// State machine for decision point
CASE eDecisionPointState OF
	E_DecisionPointState.Idle:
		bReadyStationIn[1] := FALSE;
		nDecisionPointVehicleNo := M_CTL_VehicleAtDecisionPoint();
		nDecisionPointCellNo := M_ThisCellDataIndex();
		IF (P_bTrackReady AND NOT bDecisionPoint_PAUSE) THEN
			IF ((nDecisionPointVehicleNo > 0) AND (nDecisionPointCellNo > 0) AND (nDecisionPointVehicleNo <> nLastVehicleAtDecisionPoint) ) THEN
				// New vehicle at decision point
				nLastVehicleAtDecisionPoint := nDecisionPointVehicleNo;
				// Force reading the vehicle data from track server!
				bReadDecPointVehicle := TRUE;
				// Log
				sTempString := CONCAT('TC_DP: New Vehicle NO: ', TO_STRING(nDecisionPointVehicleNo));
				IF (iCurrentTicket <> aReadCellData.stCell.astReservations[1].nTicket) THEN
					sTempString := CONCAT(sTempString, ', PriorityCount reset due to new ticket: ');
					sTempString := CONCAT(sTempString, TO_STRING(aReadCellData.stCell.astReservations[1].nTicket));
					nLastPriorityInStation := 0;
	
				END_IF
				F_LogFile(sTempString);

				eDecisionPointState := E_DecisionPointState.ReadVehicleData;
			END_IF
			IF (nDecisionPointVehicleNo = 0) THEN
				// Previous vehicle removed from DP. reset Last vehicle ID (To allow same vehicle to arrive two times!)
				nLastVehicleAtDecisionPoint := 0;
			END_IF
		END_IF
		
	E_DecisionPointState.ReadVehicleData:
		IF (NOT bReadDecPointVehicle AND NOT bReadDecPointVehicleBusy) THEN
			// Decision point vehicle data has been read!
			IF (aReadVehicleData[nDecisionPointVehicleNo].stVehicle.bDataValid) THEN
				bReadDecPointCellDone := FALSE;
				F_LogFile(CONCAT('TC_DP: Data Valid CheckTicket NO: ', TO_STRING(nDecisionPointVehicleNo)));
				eDecisionPointState := E_DecisionPointState.CheckTicket;
			ELSIF (P_bTrackReady) THEN
				F_LogFile(CONCAT('TC_DP: Data NOT valid MoveToNextCell NO: ', TO_STRING(nDecisionPointVehicleNo)));
				eDecisionPointState := E_DecisionPointState.AddExtraToList;
			ELSE
				// Disabled
				eDecisionPointState := E_DecisionPointState.Idle;
			END_IF
		END_IF			
		
	E_DecisionPointState.CheckTicket:
		// Wait to make sure cell data with reservation list has been read
		IF (bReadDecPointCellDone) THEN
			IF ( (aReadVehicleData[nDecisionPointVehicleNo].stVehicle.nTicket > 0) AND
				 (aReadCellData.stCell.astReservations[1].nTicket > 0) AND 
				 (aReadCellData.stCell.astReservations[1].nTicket = aReadVehicleData[nDecisionPointVehicleNo].stVehicle.nTicket) ) THEN
				// Ticket is OK... Save current ticket for comparison
				iCurrentTicket := aReadCellData.stCell.astReservations[1].nTicket;
				F_LogFile(CONCAT('TC_DP: Ticket Valid for this Cell. NO: ', TO_STRING(nDecisionPointVehicleNo)));
				eDecisionPointState := E_DecisionPointState.CheckPriority;
	
			ELSE
				// Ticket NOT ok for this cell
				F_LogFile(CONCAT('TC_DP: Ticket NOT Valid for this Cell. NO: ', TO_STRING(nDecisionPointVehicleNo)));
				eDecisionPointState := E_DecisionPointState.AddExtraToList;
	
			END_IF
		END_IF
		
	E_DecisionPointState.CheckPriority:
		IF (nLastPriorityInStation = (aReadVehicleData[nDecisionPointVehicleNo].stVehicle.nPriority - 1)) THEN
			// Priority is OK for this cell
			F_LogFile(CONCAT('TC_DP: Priority Valid for this Cell. NO: ', TO_STRING(nDecisionPointVehicleNo)));
			eDecisionPointState := E_DecisionPointState.TakeOwnership;

		ELSE
			// Priority is NOT ok for this cell... Keep running on highway until it macthes priority!
			F_LogFile(CONCAT('TC_DP: Priority NOT Valid for this Cell. NO: ', TO_STRING(nDecisionPointVehicleNo)));
			eDecisionPointState := E_DecisionPointState.AddExtraToList;
			
		END_IF
		
	E_DecisionPointState.TakeOwnership:
		iRes := M_CallUpdateVehicleOwner(	nVehicleID := nDecisionPointVehicleNo,
											eInputType := E_MMVehicleInputType.eMMVehicleInputType_VehicleID, 
											sInput := UINT_TO_STRING(nDecisionPointVehicleNo), 
											sCellID := sCellID 	);
		IF (iRes = 2) THEN
			// Movement call OK
			// Increase last priority
			F_LogFile(CONCAT('TC_DP: Take Ownership OK. NO: ', TO_STRING(nDecisionPointVehicleNo)));
			nLastPriorityInStation := nLastPriorityInStation + 1;
			eDecisionPointState := E_DecisionPointState.WaitStationReady;

		ELSIF (iRes = 3) THEN
			// Method call failed... Retry with the same vehicle
			// Reset Last Vehicle to accept same vehicle again
			F_LogFile(CONCAT('TC_DP: Take Ownership FAILED. NO: ', TO_STRING(nDecisionPointVehicleNo)));
			nLastVehicleAtDecisionPoint := 0;
			eDecisionPointState := E_DecisionPointState.Idle;

		END_IF		
	
	 E_DecisionPointState.WaitStationReady:
	 	// Ownership taken... Wait until station is ready for new vehicle
		IF (afbStationCtrl[1].bReadyForVehicleInput) THEN
			F_LogFile(CONCAT('TC_DP: Station ready, Veh NO: ', TO_STRING(nDecisionPointVehicleNo)));
			eDecisionPointState := E_DecisionPointState.MoveStation;

		END_IF
		
	E_DecisionPointState.MoveStation:
		//Move vehicle to station
		iRes := M_CallMoveVehicleToStationIn(	eInputType := E_MMVehicleInputType.eMMVehicleInputType_VehicleID, 
												sInput := UINT_TO_STRING(nDecisionPointVehicleNo), 
												sStationID := afbStationCtrl[1].P_sStationID,
												eDirection := E_MMDirection.eMMDirection_Forward, 
												fVelocity := 0.5, 
												fAcceleration := 1,
												iCmdID => iDecisionPointMoveCmdID 	);
	
		IF (iRes = 2) THEN
			// Movement call OK
			stVehicleOnStation := aReadVehicleData[nDecisionPointVehicleNo];
			eDecisionPointState := E_DecisionPointState.WaitMoveStation;

		ELSIF (iRes = 3) THEN
			// Movement call failed... Try again with same vehicle
			nLastVehicleAtDecisionPoint := 0;
			nLastPriorityInStation := nLastPriorityInStation - 1;	// Go back to previous priority
			F_LogFile(CONCAT('TC_DP: Move to station FAILED, Veh NO: ', TO_STRING(nDecisionPointVehicleNo)));
			eDecisionPointState := E_DecisionPointState.Idle;

		END_IF
		
(*	E_DecisionPointState.WaitMoveStation:
		IF (aReadVehicleData[nDecisionPointVehicleNo].stVehicle.sCurrentStationID = aStations[1].sStationID) THEN
			bReadyStationIn := TRUE;
			F_LogFile(CONCAT('TC_DP: Wait station reached, Veh NO: ', TO_STRING(nDecisionPointVehicleNo)));
			
			IF ((aReadVehicleData[nDecisionPointVehicleNo].stVehicle.bDataValid) AND  
				(nLastPriorityInStation = aReadVehicleData[nDecisionPointVehicleNo].stVehicle.nTicketSize) ) THEN
				// Last vehicle in ticket handled... Remove reservation
				iTicketToRemove := aReadVehicleData[nDecisionPointVehicleNo].stVehicle.nTicket;
				eDecisionPointState := E_DecisionPointState.RemoveReservation;

			ELSE
				eDecisionPointState := E_DecisionPointState.Idle;

			END_IF
			
		END_IF
*)		
	E_DecisionPointState.WaitMoveStation:
		tonDecisionPointDelay.IN := TRUE;
		tonDecisionPointDelay.PT := T#1S;
		IF (tonDecisionPointDelay.Q) THEN
			iRes := M_CallMoveVehicleStatus(iCommandID := iDecisionPointMoveCmdID,
											eMoveStatus => eDecisionPointMoveState 	);
			IF (iRes = 2) THEN
				tonDecisionPointDelay.IN := FALSE;
				// Trig event-driven reading
				M_VehicleToReadAdd(nDecisionPointVehicleNo);
				// Call completed... Check move status
				IF (eDecisionPointMoveState >= E_VehicleMoveState.ErrorLocation) THEN
					// TODO!!! - Error during movement
					
				ELSIF (eDecisionPointMoveState = E_VehicleMoveState.Complete) THEN
					// Movement completed
					bReadyStationIn[1] := TRUE;
					
					IF ((aReadVehicleData[nDecisionPointVehicleNo].stVehicle.bDataValid) AND  
						(nLastPriorityInStation = aReadVehicleData[nDecisionPointVehicleNo].stVehicle.nTicketSize) ) THEN
						// Last vehicle in ticket handled... Remove reservation
						iTicketToRemove := aReadVehicleData[nDecisionPointVehicleNo].stVehicle.nTicket;
						eDecisionPointState := E_DecisionPointState.RemoveReservation;
		
					ELSE
						eDecisionPointState := E_DecisionPointState.Idle;
		
					END_IF					
					F_LogFile(CONCAT('TC_DP: Wait station reached, Veh NO: ', TO_STRING(nDecisionPointVehicleNo)));
					
				END_IF
				
			ELSIF (iRes = 3) THEN
				// TODO!!!
				// Try again
				tonDecisionPointDelay(IN := FALSE);
				// Trig event-driven reading
				M_VehicleToReadAdd(nDecisionPointVehicleNo);
				
			END_IF
			
		END_IF

	E_DecisionPointState.RemoveReservation:
		// Check if the specified ticket is expected at the specified station
		iRes := M_CallRemoveReservation(sStationID:= afbStationCtrl[1].P_sStationID, nTicket:= iTicketToRemove);
			
		IF (iRes = 2) THEN
			// Movement call OK
			nLastPriorityInStation := 0;
			F_LogFile(CONCAT('TC_DP: Removed ticket reservation OK NO: ', TO_STRING(iTicketToRemove)));
			eDecisionPointState := E_DecisionPointState.Idle;

		ELSIF (iRes = 3) THEN
			// Movement call failed
			// TODO!!!
			F_LogFile(CONCAT('TC_DP: Remove ticket reservation FAILED NO: ', TO_STRING(nDecisionPointVehicleNo)));
			eDecisionPointState := E_DecisionPointState.Idle;
			
		END_IF
		
	E_DecisionPointState.AddExtraToList:
		// Add this vehicle to the list of surveilled vehicles
		IF ( M_ExtraVehicleAdd(nDecisionPointVehicleNo) ) THEN
			F_LogFile(CONCAT('TC_DP: Added to extra list without ownership. NO: ', TO_STRING(nDecisionPointVehicleNo)));
			eDecisionPointState := E_DecisionPointState.WaitStationEmpty;
			
		END_IF
	 
	E_DecisionPointState.WaitStationEmpty:
		IF (bStationEmpty) THEN
			// Not for this station and device is empty
			F_LogFile(CONCAT('TC_DP: Station Empty. veh. NO: ', TO_STRING(nDecisionPointVehicleNo)));
			eDecisionPointState := E_DecisionPointState.MoveNextCell;

		END_IF	
		
	E_DecisionPointState.MoveNextCell:
		IF ((nVehicleNoToRemove > 0) AND (nDecisionPointVehicleNo = nVehicleNoToRemove)) THEN
			// Remove the vehicle number
			iRes := M_CallMoveVehicleToPosition(eInputType := E_MMVehicleInputType.eMMVehicleInputType_VehicleID,
												sInput := UINT_TO_STRING(nDecisionPointVehicleNo),
												nPathID := 17,
												fPosition := 0.3, 
												eDirection := E_MMDirection.eMMDirection_Forward, 
												fVelocity := 1,
												fAcceleration := 1 	);
			IF (iRes = 2) THEN
				// Movement call OK
				nVehicleNoToRemove := 0;
				F_LogFile(CONCAT('TC_DP: Moved vehicle to track out: ', TO_STRING(nDecisionPointVehicleNo)));
				eDecisionPointState := E_DecisionPointState.Idle;
				
			ELSIF (iRes = 3) THEN
				// Movement call failed... Retry with same vehicle
				F_LogFile(CONCAT('TC_DP: Error Moving to track out: ', TO_STRING(nDecisionPointVehicleNo)));
				nLastVehicleAtDecisionPoint := 0;
				eDecisionPointState := E_DecisionPointState.Idle;
				
			END_IF
		ELSE			
			//Move vehicle to station 2  - which will send to next cell
			iRes := M_CallMoveVehicleToStationIn(	eInputType := E_MMVehicleInputType.eMMVehicleInputType_VehicleID, 
													sInput := UINT_TO_STRING(nDecisionPointVehicleNo), 
													sStationID := afbStationCtrl[2].P_sStationID,
													eDirection := E_MMDirection.eMMDirection_Forward, 
													fVelocity := 0.5, 
													fAcceleration := 1,
													iCmdID => iDecisionPointMoveCmdID 	);

			IF (iRes = 2) THEN
				// Movement call OK
				// Trig event-driven reading
				M_VehicleToReadAdd(nDecisionPointVehicleNo);				
				eDecisionPointState := E_DecisionPointState.WaitMoveNextCell;
				
			ELSIF (iRes = 3) THEN
				// Movement call failed... Try again with same vehicle
				nLastVehicleAtDecisionPoint := 0;
				F_LogFile(CONCAT('TC_DP: Move to next station FAILED NO: ', TO_STRING(nDecisionPointVehicleNo)));
				eDecisionPointState := E_DecisionPointState.Idle;
				
			END_IF
		END_IF

	E_DecisionPointState.WaitMoveNextCell:
		tonDecisionPointDelay.IN := TRUE;
		tonDecisionPointDelay.PT := T#1S;
		IF (tonDecisionPointDelay.Q) THEN
			iRes := M_CallMoveVehicleStatus(	iCommandID := iDecisionPointMoveCmdID,
												eMoveStatus => eDecisionPointMoveState 	);
		
			IF (iRes = 2) THEN
				tonDecisionPointDelay.IN := FALSE;
				// Call OK
				IF (eDecisionPointMoveState >= E_VehicleMoveState.ErrorLocation) THEN
					// Error with command
					// TODO!!!
					
				ELSIF (eDecisionPointMoveState >= E_VehicleMoveState.Accepted) THEN
					// Command accepted!
					F_LogFile(CONCAT('TC_DP: Vehicle moved to next cell: ', TO_STRING(nDecisionPointVehicleNo)));
					eDecisionPointState := E_DecisionPointState.Idle;			
					
				END_IF
				
			ELSIF (iRes = 3) THEN
				tonDecisionPointDelay.IN := FALSE;
				// Movement call failed... Retry with same vehicle
				nLastVehicleAtDecisionPoint := 0;
				eDecisionPointState := E_DecisionPointState.Idle;
				
			END_IF

		END_IF

END_CASE

tonDecisionPointDelay(	IN:= ,
						PT:= ,
						Q=> ,
						ET=> );
END_METHOD

METHOD PROTECTED M_CTL_ExitPoint : BOOL
VAR_INPUT
END_VAR
VAR
	iRes				: INT;
END_VAR
VAR 
END_VAR
// State machine for exit point
CASE eExitPointState OF
	E_ExitPointState.Idle:
		tonExitPointDelay.IN := FALSE;
		IF (bEnable) THEN
			eExitPointState := E_ExitPointState.CheckBuffer;
		END_IF

	E_ExitPointState.CheckBuffer:
		M_CTL_CheckStationsPostBuffer(iTicket => iExitPointTicket, iStationID => iExitPointStation, iBufferIndex => iExitPointFirstIdx);
		IF (iExitPointStation > 0) THEN
			IF ( (iExitPointTicket > 0) AND (iExitPointFirstIdx > 0) ) THEN
								
				tonExitPointDelay.IN := TRUE;
				tonExitPointDelay.PT := TO_TIME(stAdditionalDataIn.ExitPointReleaseDelay * 1000.0);
				//Delay before releasing a ticket for tickets size of 3 vehicles

				IF (tonExitPointDelay.Q) THEN
					tonExitPointDelay.IN := FALSE;
					// A station is ready to deliver from post buffer
					iExitPointBufferIdx := MM_MAX_BUFFER_INDEX;
					F_LogLine(CONCAT('TC_EP: Ticket ready at EP (%d) from idx: ', UINT_TO_STRING(iExitPointFirstIdx)), iExitPointTicket);
					IF stTrafficLightLocation.fPosition > 0 THEN //Traffic light on cell?
						eExitPointState := E_ExitPointState.SetTrafficLightRd;
					ELSE
						eExitPointState := E_ExitPointState.WaitVehicleOnPos;
					END_IF
					
					//Special for this cell. Ready station flags used to handle shoes in right order and are not lowered until now.
					bReadyStationIn[1] := FALSE;
					bReadyStationIn[2] := FALSE;
					bReadyStationOut[2] := FALSE;
				END_IF
				
			ELSIF (afbBufferControlPost[iExitPointStation].P_iCurrentVehicleID > 0 AND afbBufferControlPost[iExitPointStation].P_iCurrentVehicleTicket = 0) THEN
				 F_LogLine(CONCAT('TC_EP: Ticket MISSING for vehicle at EP (%d) from idx: ', UINT_TO_STRING(iExitPointFirstIdx)), iExitPointTicket);
			
				IF stTrafficLightLocation.fPosition > 0 THEN //Traffic light on cell?
					eExitPointState := E_ExitPointState.SetTrafficLightRd;
				ELSE
					eExitPointState := E_ExitPointState.WaitVehicleOnPos;
				END_IF
				
				//Special for this cell. Ready station flags used to handle shoes in right order and are not lowered until now.
				bReadyStationIn[1] := FALSE;
				bReadyStationIn[2] := FALSE;
				bReadyStationOut[2] := FALSE;
			END_IF
		END_IF
	
	E_ExitPointState.SetTrafficLightRd:
		iRes := M_CallSetTrafficLightColor(	nTrafficLightNo := 1,
											nColor := E_MMTrafficLightColor.eMMTrafficLightColor_Red );
		IF (iRes = 2) THEN
			// Call OK
			F_LogLine('TC_EP: TL set to red OK', 0);
			eExitPointState := E_ExitPointState.TrafficLightRedDelay;
		ELSIF (iRes = 3) THEN
			// Call failed
			// TODO!!!
			F_LogLine('TC_EP: Error setting TL to red', 0);
			eExitPointState := E_ExitPointState.TrafficLightRedDelay;
		END_IF
	
	E_ExitPointState.TrafficLightRedDelay:
		tonExitPointDelay.IN := TRUE;
		tonExitPointDelay.PT := T#3S;
		IF (tonExitPointDelay.Q) THEN
			tonExitPointDelay.IN := FALSE;
			eExitPointState := E_ExitPointState.WaitVehicleOnPos;			
		END_IF
		
	E_ExitPointState.WaitVehicleOnPos:
		// Wait for vehicle to be on position
		iExitPointVehicleID := afbBufferControlPost[iExitPointStation].P_iCurrentVehicleID;
		iExitPointMoveCmdID := afbBufferControlPost[iExitPointStation].P_iCurrentVehicleCmdID;
		
		tonExitPointDelay.IN := TRUE;
		tonExitPointDelay.PT := T#1S;
		IF (tonExitPointDelay.Q) THEN
			iRes := M_CallMoveVehicleStatus(iCommandID := iExitPointMoveCmdID,
												eMoveStatus => eExitPointMoveState 	);
			
				IF (iRes = 2) THEN
					tonExitPointDelay.IN := FALSE;
					// Call OK
					IF (eExitPointMoveState >= E_VehicleMoveState.ErrorLocation) THEN
						// Error with command
						// TODO!!!
						
					ELSIF (eExitPointMoveState >= E_VehicleMoveState.Complete) THEN
						// Command accepted!
						F_LogLine('TC_EP: Vehicle on buffer out: (%d)', iExitPointVehicleID);
						eExitPointState := E_ExitPointState.MoveVehicle;
					END_IF
					
				ELSIF (iRes = 3) THEN
					tonExitPointDelay.IN := FALSE;
					// Movement call failed... Retry with same vehicle
					eExitPointState := E_ExitPointState.Done;
				END_IF
			END_IF
	
	E_ExitPointState.MoveVehicle:
		//Move vehicle from last position in buffer
		iRes := M_CallMoveVehicleToDecisionPoint(eInputType := E_MMVehicleInputType.eMMVehicleInputType_VehicleID, 
													 sInput := UINT_TO_STRING(iExitPointVehicleID), 
													 sStationID := sNextStationOnTrack,
													 eDirection := E_MMDirection.eMMDirection_Forward, 
													 fVelocity := 1, 
													 fAcceleration := 1	);
													 
			 IF (iRes = 2) THEN
				// Movement call OK
				// Read vehicle data
				M_VehicleToReadAdd(iExitPointVehicleID);
				F_LogLine('TC_EP: Vehicle moved from Post-Buf (%d)', iExitPointVehicleID);
				afbBufferControlPost[iExitPointStation].M_RemoveVehicle(iVehicleID:= iExitPointVehicleID);
				
				// More vehicles in buffer?
				IF afbBufferControlPost[iExitPointStation].M_IsEmpty() THEN
					F_LogLine(CONCAT('TC_EP: Vehicle on buffer moving out, buffer empty: %d', UINT_TO_STRING(iExitPointFirstIdx)), iExitPointTicket);
					eExitPointState := E_ExitPointState.WaitMoveVehicle;
				ELSE
					IF afbBufferControlPost[iExitPointStation].P_iCurrentVehicleTicket <> iExitPointTicket THEN
						F_LogLine(CONCAT('TC_EP: Vehicle on buffer moving out, New ticket: %d', UINT_TO_STRING(iExitPointFirstIdx)), iExitPointTicket);
						eExitPointState := E_ExitPointState.WaitMoveVehicle;
					ELSE
						F_LogLine(CONCAT('TC_EP: Vehicle on buffer moving out, more vehicles: %d', UINT_TO_STRING(iExitPointFirstIdx)), iExitPointTicket);
						eExitPointState := E_ExitPointState.WaitVehicleOnPos;	
					END_IF
				END_IF
				
			ELSIF (iRes = 3) THEN
				// Movement call failed
				// TODO!!!
				F_LogLine('TC_EP: Failed moving vehicle moved from Post-Buf (%d)', iExitPointVehicleID);
				F_LogLine(CONCAT('Message: ', WSTRING_TO_STRING(stMoveToDecisionPointData.stOutput.sMessage)), 0); 
				IF stTrafficLightLocation.fPosition > 0 THEN //Traffic light on cell?
					eExitPointState := E_ExitPointState.SetTrafficLightGr;
				ELSE
					eExitPointState := E_ExitPointState.Done;
				END_IF
			END_IF
			
	E_ExitPointState.WaitMoveVehicle:
		tonExitPointDelay.IN := TRUE;
		tonExitPointDelay.PT := T#60S;
		M_VehicleToReadAdd(iExitPointVehicleID);
		IF ((tonExitPointDelay.ET > T#0S)) THEN
			IF (aReadVehicleData[iExitPointVehicleID].stVehicle.nPathID <> aStations[iExitPointStation].stStationData1.stLocation.nPathID) THEN
				F_LogLine('TC_EP: Vehicle moved from path set green light (%d)', aStations[iExitPointStation].astPostBuffer[iExitPointBufferIdx].nCurrentVehicleID);
				IF stTrafficLightLocation.fPosition > 0 THEN //Traffic light on cell?
					eExitPointState := E_ExitPointState.SetTrafficLightGr;
				ELSE
					eExitPointState := E_ExitPointState.Done;
				END_IF
			END_IF
		END_IF
		
	E_ExitPointState.SetTrafficLightGr:
		IF stTrafficLightLocation.fPosition > 0 THEN //Traffic light on cell?
			iRes := M_CallSetTrafficLightColor(	nTrafficLightNo := 1,
												nColor := E_MMTrafficLightColor.eMMTrafficLightColor_Green );
			IF (iRes = 2) THEN
				// Call OK
				F_LogLine('TC_EP: TL set to green OK', 0);
				eExitPointState := E_ExitPointState.Idle;
			ELSIF (iRes = 3) THEN
				// Call failed
				F_LogLine('TC_EP: Error setting TL to green', 0);
				eExitPointState := E_ExitPointState.Idle;
			END_IF
		ELSE
			eExitPointState := E_ExitPointState.Done;
		END_IF
		
	E_ExitPointState.Done:
		eExitPointState := E_ExitPointState.Idle;
	
END_CASE

// Delay
tonExitPointDelay(	IN:= ,
					PT:= ,
					Q=> ,
					ET=> 	);
END_METHOD

METHOD M_CTL_Station : BOOL
VAR_INPUT
END_VAR
VAR
	iRes				: INT;
	sTempString			: STRING(200);
	i					: UINT;
END_VAR
IF bVehicleMovedFromSt1 THEN
	aStations[1].stStationData1.nReservedVehicleID := 0;
	aStations[1].stStationData1.nCurrentVehicleID := 0;
	aStations[1].stStationData1.nTicket := 0;
	aStations[1].stStationData1.nTicketSize := 0;
	aStations[1].stStationData1.CurrentPriority := 0;
	bVehicleMovedFromSt1 := FALSE;
END_IF


iVehicleReadyStation1 := M_CTL_VehicleAtStationX(iStationNo:= 1);
iVehicleReadyStation2 := M_CTL_VehicleAtStationX(iStationNo:= 2);

//Run stateTimers
IF bStationStateChangeOS THEN
	diStationStateTimer := 0;
END_IF
IF diStationStateTimer < 64000 THEN
	diStationStateTimer := diStationStateTimer + g_iPLCScan_MS;
END_IF

//Station 2 sequence
CASE eStationState OF
	E_StationState.Idle:
		IF (P_bTrackReady) THEN
			bVehicleFoundCmdBuffer := FALSE;
			eStationState := E_StationState.CheckStations;
		END_IF
		
	E_StationState.CheckStations:
		IF ( (iVehicleReadyStation2 > 0) AND (iVehicleReadyStation2 <> nLastVehicleAtStation2) ) THEN
			iVehicleMoveBufferIN := iVehicleReadyStation2;
			sTempString := CONCAT('TC_STAT2: Vehicle NO: ', TO_STRING(iVehicleReadyStation2));
			F_LogFile(CONCAT(sTempString, ', Ready out'));
			
			// Check if post buffer is activated
			IF (aStations[2].astPostBuffer[1].bPresent) THEN
				// Use post buffer
				IF (aStations[2].stStationData1.bPresent AND ((iVehicleMoveBufferIN > 0) AND (iVehicleMoveBufferIN <= MM_MAX_NUMBER_OF_VEHICLE_ELEMENTS))) THEN
					// Update station data with correct values
					aStations[2].stStationData1.nReservedVehicleID := iVehicleMoveBufferIN;
					aStations[2].stStationData1.nCurrentVehicleID := iVehicleMoveBufferIN;
					aStations[2].stStationData1.nTicket := aReadVehicleData[iVehicleMoveBufferIN].stVehicle.nTicket;
					aStations[2].stStationData1.nTicketSize := aReadVehicleData[iVehicleMoveBufferIN].stVehicle.nTicketSize;
					aStations[2].stStationData1.CurrentPriority := aReadVehicleData[iVehicleMoveBufferIN].stVehicle.nPriority;
					// Log
					F_LogFile('Send to post buffer');
					// Signal that vehicle can be moved from station
					afbStationCtrl[2].bCompletedInput := TRUE;
					eStationState := E_StationState.MoveToPostBuf;
	
				END_IF
			ELSE
				// No post buffer on this station, send directly to next cell
				F_LogFile('Send to next cell');
				eStationState := E_StationState.MoveToNextCell;
				
			END_IF
			// JLH_21.11.16: Test - To make sure vehicle is removed form FIFO!
			P_iVehicleFifoOut := iVehicleMoveBufferIN;

		ELSIF (NOT P_bTrackReady) THEN
			// Disabled!
			eStationState := E_StationState.Idle;

		END_IF
		IF (iVehicleReadyStation2 = 0) THEN
			// Previous vehicle removed from ST2. Reset Last vehicle ID (To allow same vehicle to arrive two times!)
			nLastVehicleAtStation2 := 0;

		END_IF
	
	E_StationState.MoveToPostBuf:
		IF (aStations[2].stStationData1.nCurrentVehicleID <> iVehicleMoveBufferIN) THEN
			P_iVehicleFifoOut := iVehicleMoveBufferIN;
			afbStationCtrl[2].bCompletedInput := FALSE;
			eStationState := E_StationState.Idle;
			
		END_IF
	
	E_StationState.MoveToNextCell:
		iRes := M_CallMoveVehicleToDecisionPoint(	eInputType := E_MMVehicleInputType.eMMVehicleInputType_VehicleID, 
//												 	sInput := UINT_TO_STRING(iVehicleReadyStation2), 
												 	sInput := UINT_TO_STRING(iVehicleMoveBufferIN), 
												 	sStationID := sNextStationOnTrack,
												 	eDirection := E_MMDirection.eMMDirection_Forward, 
												 	fVelocity := 1, 
													fAcceleration := 1,
													iCmdId => iStation2MoveCmdID 	);
		IF (iRes = 2) THEN
			// Movement call OK
			sTempString := CONCAT('TC_STAT2: Move vehicle call: ', TO_STRING(iVehicleMoveBufferIN));
			F_LogFile(CONCAT(sTempString, ', out OK'));
			eStationState := E_StationState.ExtraVehicleRemove;

		ELSIF (iRes = 3) THEN
			// Movement call failed... Retry with same vehicle
			sTempString := CONCAT('TC_STAT2: Move vehicle call: ', TO_STRING(iVehicleMoveBufferIN));
			F_LogFile(CONCAT(sTempString, ', out Failed'));
			F_LogFile(CONCAT(' - Error message: ', TO_STRING(stMoveToDecisionPointData.stOutput.sMessage)));
			// reset last vehicle to make sure it will handle it again!
			nLastVehicleAtStation2 := 0;
			eStationState := E_StationState.Idle;
			
		END_IF
				
	E_StationState.ExtraVehicleRemove:
		// Remove the vehicle from the list of vehicles to be surveilled
		IF (M_ExtraVehicleRemove(iVehicleNo:= iVehicleMoveBufferIN)) THEN
			F_LogFile(CONCAT('TC_STAT2: Vehicle removed from extra, NO: ', TO_STRING(iVehicleMoveBufferIN)));
			eStationState := E_StationState.AddReservation;
			
		ELSE
			F_LogFile(CONCAT('TC_STAT2: Vehicle NOT removed from extra, NO: ', TO_STRING(iVehicleMoveBufferIN)));
			eStationState := E_StationState.AddReservation;
		
		END_IF
	
	E_StationState.AddReservation:
		//Speciel handling for this cell - find and addReservation for this vehicle based on command data in buffer
		IF NOT bVehicleFoundCmdBuffer THEN
			FOR i:=0 TO 10 DO
				IF M_CarrierIDToVehicleID(arVehicleCommandBuffer[i].CarrierID) = iVehicleMoveBufferIN THEN
					bVehicleFoundCmdBuffer := TRUE;
					bVehicleCmdPointer := i;
					EXIT;
				END_IF		
			END_FOR
			
			IF NOT bVehicleFoundCmdBuffer THEN
				F_LogLine('TC_EP: WARNING Command data NOT found in buffer, VehicleID: %d', TO_UINT(iVehicleMoveBufferIN));
				eStationState := E_StationState.Done;
			END_IF
		END_IF
		
		IF bVehicleFoundCmdBuffer THEN
			iRes := M_CallAddReservation(	sStationID := arVehicleCommandBuffer[bVehicleCmdPointer].TargetStation,
											sCarrierID := arVehicleCommandBuffer[bVehicleCmdPointer].CarrierID,
											nTicket := arVehicleCommandBuffer[bVehicleCmdPointer].Ticket,
											nTicketSize := arVehicleCommandBuffer[bVehicleCmdPointer].CarriersInPackage,
											nPriority := arVehicleCommandBuffer[bVehicleCmdPointer].Priority 	);
			IF (iRes = 2) THEN
				// Success
				MEMSET(ADR(arVehicleCommandBuffer[bVehicleCmdPointer]), 0, SIZEOF(arVehicleCommandBuffer[bVehicleCmdPointer]));
				F_LogLine('TC_EP: Command data deleted from buffer, VehicleID: %d', TO_UINT(iVehicleMoveBufferIN));
				eStationState := E_StationState.Done;
			ELSIF (iRes = 3) THEN
				// Error!
				F_LogLine('TC_EP: AddReservation failed, VehicleID: %d', TO_UINT(iVehicleMoveBufferIN));
				eStationState := E_StationState.Done;
			END_IF
		END_IF	

	E_StationState.Done:
		nLastVehicleAtStation2 := iVehicleMoveBufferIN;
		sTempString := CONCAT('TC_STAT2: Move vehicle: ', TO_STRING(iVehicleMoveBufferIN));
		F_LogFile(CONCAT(sTempString, ', State done'));
		eStationState := E_StationState.Idle;

END_CASE

//OS state Change
bStationStateChangeOS := eStationState <> eStationState_Old;
eStationState_Old := eStationState;
END_METHOD

/// Returns the Vehicle ID of the vehicle at the station decision point (0 if no vehicle ready)
METHOD M_CTL_VehicleAtDecisionPoint : UINT
VAR_INPUT
END_VAR
VAR
	iCellNo		: UINT;
	
	iStationNo	: UINT;
END_VAR

// Get cell number/index
iCellNo := M_ThisCellDataIndex();

(* OLD!
IF (iCellNo > 0) THEN
	// Check Cell ID
	IF (aReadCellData.stCell.nVehicleIDDecisionPoint > 0) THEN
//		IF (aReadCellData.stCell.nVehicleIDDecisionPoint <> nLastVehicleAtDecisionPoint) THEN
			// New vehicle arrived at decision point
			M_CTL_VehicleAtDecisionPoint := aReadCellData.stCell.nVehicleIDDecisionPoint;
			RETURN;
//		END_IF
		M_CTL_VehicleAtDecisionPoint := 0;
	END_IF
	M_CTL_VehicleAtDecisionPoint := 0;
END_IF
*)

 //NEW - One decision point FOR each station
IF (iCellNo > 0) THEN
	iStationNo := 1;
	WHILE (iStationNo <= MM_MAX_NUMBER_OF_STATION_ELEMENTS) DO
	// Find correct station data
	// NOTE! only one station in this cell
		IF (aReadStationData[iStationNo].stStationData.sStationID = aStations[1].sStationID) THEN
			// Find first vehicle at station decision point
			IF (aReadStationData[iStationNo].stStationData.nVehicleIDDecisionPoint > 0) THEN
				M_CTL_VehicleAtDecisionPoint := aReadStationData[iStationNo].stStationData.nVehicleIDDecisionPoint;
				RETURN;
			END_IF
		END_IF
		iStationNo := iStationNo + 1;
	END_WHILE
END_IF


// None found
M_CTL_VehicleAtDecisionPoint := 0;
END_METHOD

/// Returns the Vehicle ID of the vehicle at the station x defined on input (0 if no vehicle)
METHOD M_CTL_VehicleAtStationX : UINT
VAR_INPUT
	iStationNo	: UINT;
END_VAR
VAR
	iCellNo		: UINT;
	i			: UINT;
END_VAR
// Get cell number/index
iCellNo := M_ThisCellDataIndex();

IF (iCellNo > 0) THEN
	i := 1;
	WHILE (i <= MM_MAX_NUMBER_OF_STATION_ELEMENTS) DO
	// Find correct station data
		IF (aReadStationData[i].stStationData.sStationID = aStations[iStationNo].sStationID) THEN
			// Find vehicle at station x
			IF (aReadStationData[i].stStationData.nVehicleIDStationIn > 0) THEN
				M_CTL_VehicleAtStationX := aReadStationData[i].stStationData.nVehicleIDStationIn;
				RETURN;
			END_IF
		END_IF
		i := i + 1;
	END_WHILE
END_IF


// None found
M_CTL_VehicleAtStationX := 0;
END_METHOD

// Set data for traffic light
METHOD PUBLIC M_DefineStation : BOOL
VAR_INPUT
	nStationNo			: UINT(1..5);
	sStationID			: STRING(30);
	nLoc1PathID			: UINT;		// Path number for input location
	rLoc1Position		: REAL;		// Distance on the specified path for input location
	nLoc2PathID			: UINT;		// Path number for output location (0 if single station)
	rLoc2Position		: REAL;		// Distance on the specified path for output location (0.0 if single station)
	nLocDecPathID		: UINT;		// Path number for decision point location
	rLocDecPosition		: REAL;		// Distance on the specified path for decision point location
	nPreBufferSize		: UINT;		// Size of pre buffer (number of positions)
	nPostBufferSize		: UINT;		// Size of post buffer (number of positions)
END_VAR
VAR
END_VAR

// Call Base class method and add data to BufferControl FB's if it returns TRUE
IF (SUPER^.M_DefineStation(	nStationNo := nStationNo,
							sStationID := sStationID,
							nLoc1PathID := nLoc1PathID,
							rLoc1Position := rLoc1Position,
							nLoc2PathID := nLoc2PathID,
							rLoc2Position := rLoc2Position,
							nLocDecPathID := nLocDecPathID,
							rLocDecPosition := rLocDecPosition,
							nPreBufferSize := nPreBufferSize,
							nPostBufferSize := nPostBufferSize)) THEN

	//Set buffersize and type in BufferControl
	afbBufferControlPre[nStationNo].P_iBufferSize := nPreBufferSize;
	afbBufferControlPost[nStationNo].P_iBufferSize := nPostBufferSize;
	afbBufferControlPre[nStationNo].P_sBufferType := 'Pre';
	afbBufferControlPost[nStationNo].P_sBufferType := 'Post';
	
	M_DefineStation := TRUE;

ELSE
	M_DefineStation := FALSE;

END_IF
END_METHOD

METHOD PROTECTED M_Init : BOOL
VAR_INPUT
END_VAR
VAR
	i : UINT;
	sTemp : STRING;
END_VAR

M_Init := SUPER^.M_Init();
END_METHOD

METHOD PROTECTED M_Run : BOOL
VAR_INPUT
END_VAR
VAR
	i	: USINT;
END_VAR

// Call base class FB
// Handles method calls to trackserver and status data reading from trackserver
SUPER^.M_Run();

///////////////////////////////////////////////////////////////////////////////////////////////////////////////////
// FB's for Station data handling
///////////////////////////////////////////////////////////////////////////////////////////////////////////////////
afbStationCtrl[1].bCompletedInput := abStation1Done[1];
afbStationCtrl[1].bCompletedOutput := abStation2Done[1];
afbStationCtrl[1](stStationData := aStations[1]);
afbStationCtrl[2].bCompletedInput := abStation1Done[2];
afbStationCtrl[2].bCompletedOutput := abStation2Done[2];
afbStationCtrl[2](stStationData := aStations[2]);
afbStationCtrl[3].bCompletedInput := abStation1Done[3];
afbStationCtrl[3].bCompletedOutput := abStation2Done[3];
afbStationCtrl[3](stStationData := aStations[3]);
afbStationCtrl[4].bCompletedInput := abStation1Done[4];
afbStationCtrl[4].bCompletedOutput := abStation2Done[4];
afbStationCtrl[4](stStationData := aStations[4]);
afbStationCtrl[5].bCompletedInput := abStation1Done[5];
afbStationCtrl[5].bCompletedOutput := abStation2Done[5];
afbStationCtrl[5](stStationData := aStations[5]);

//New buffer handling
		FOR i := 1 TO 5 DO
			afbBufferControlPre[i](stMMBuffer:= aStations[i].astPreBuffer);
			afbBufferControlPost[i](stMMBuffer:= aStations[i].astPostBuffer);
		END_FOR
END_METHOD

PROPERTY P_bStationEmpty : BOOL
SET
bStationEmpty := P_bStationEmpty;
END_SET
END_PROPERTY

PROPERTY P_bVehicleMovedFromSt1 : BOOL
GET
P_bVehicleMovedFromSt1 := bVehicleMovedFromSt1;
END_GET
SET
bVehicleMovedFromSt1 := P_bVehicleMovedFromSt1;
END_SET
END_PROPERTY

PROPERTY P_CarriersFIFO : ARRAY[1..10] OF ST_VehicleInHS
GET // PUBLIC
P_CarriersFIFO := aVehiclesStationFIFO;
END_GET
SET // PUBLIC
aVehiclesStationFIFO := P_CarriersFIFO;
END_SET
END_PROPERTY

PROPERTY PUBLIC P_eTrafficLightColor : E_MMTrafficLightColor
GET
P_eTrafficLightColor := stTrafficLightColorData.stOutput.nTrafficLightColor;
END_GET
END_PROPERTY

PROPERTY P_iVehicleFifoOut : UINT
GET
P_iVehicleFifoOut := iVehicleFIFOOut;
END_GET
SET
iVehicleFIFOOut := P_iVehicleFifoOut;
END_SET
END_PROPERTY

PROPERTY P_StationEmptyReady : BOOL
SET
afbStationCtrl[1].bReadyForVehicleInput := P_StationEmptyReady;
END_SET
END_PROPERTY

PROPERTY P_stReservation : ST_ReservationData
GET
P_stReservation := aReadCellData.stCell.astReservations[1];
END_GET
END_PROPERTY

PROPERTY PUBLIC P_stVehicleDataOnStation : ST_ReadVehicleData
GET
P_stVehicleDataOnStation := stVehicleOnStation;
END_GET
END_PROPERTY

END_FUNCTION_BLOCK

// ---- ECC/Basic/TrackClient/FB_TrackClient_Basic.TcPOU
FUNCTION_BLOCK FB_TrackClient_Basic
VAR_INPUT
	bEnable			: BOOL;
	bEStopOK		: BOOL;
	bSuspend		: BOOL;
	bReset			: BOOL;
	abStation1Ready	: ARRAY [1..5] OF BOOL;	// TRUE when station is ready for a vehicle at input
	abStation2Ready	: ARRAY [1..5] OF BOOL; // TRUE when station is ready for a vehicle at output
	abStation1Done	: ARRAY [1..5] OF BOOL;	// TRUE when station picked up last from vehicle at input
	abStation2Done	: ARRAY [1..5] OF BOOL; // TRUE when station placed last at vehicle at output
	abStation1ReworkReq	: ARRAY [1..5] OF BOOL;	// TRUE when station signals that rework is needed for carrier at station 1 (input) 
	abStation2ReworkReq	: ARRAY [1..5] OF BOOL;	// TRUE when station signals that rework is needed for carrier at station 2 (output)
	abStation1ReworkDone: ARRAY [1..5] OF BOOL;	// TRUE when station signals that rework is done for carrier at station 1 (input) 
	abStation2ReworkDone: ARRAY [1..5] OF BOOL;	// TRUE when station signals that rework is done for carrier at station 2 (output)
END_VAR
VAR_OUTPUT
	{attribute 'OPC.UA.DA':='1'}
	{attribute 'OPC.UA.DA.Access' := '1'}
	{attribute 'OPC.UA.DA.Description' := 'TRUE if connected to call methods on Track server'}
	{attribute 'OPC.UA.DA.DisplayName' := 'TRUE if connected to call methods on Track server'}
	bConnectedMethod: BOOL;
	{attribute 'OPC.UA.DA':='1'}
	{attribute 'OPC.UA.DA.Access' := '1'}
	{attribute 'OPC.UA.DA.Description' := 'TRUE if connected for data reading from Track Server'}
	{attribute 'OPC.UA.DA.DisplayName' := 'TRUE if connected for data reading from Track Server'}
	bConnectedNode	: BOOL;
	{attribute 'OPC.UA.DA':='1'}
	{attribute 'OPC.UA.DA.Access' := '1'}
	{attribute 'OPC.UA.DA.Description' := 'TRUE if cell info is created on track server'}
	{attribute 'OPC.UA.DA.DisplayName' := 'TRUE if cell info is created on track server'}
	bTrackInitDone	: BOOL;
	{attribute 'OPC.UA.DA':='0'}
	bBusyMethod		: BOOL;
	bVehicleInitDone: BOOL;
	bErrorMethod	: BOOL;
	nErrorMethodID	: E_OPC_UA_Errors;
	bErrorNode		: BOOL;
	nErrorNodeID	: E_OPC_UA_Errors;
	bStarted		: BOOL;
	bSuspended		: BOOL;
	bReadyStationIn	: ARRAY [1..5] OF BOOL;
	bReadyStationOut: ARRAY [1..5] OF BOOL;
	stErrorWarning	: ST_OutputErrorWarning;
END_VAR
VAR_IN_OUT
	// Inputs
	stCommand		: ST_InputTransportCommand;
	stMappingIn		: ST_InputTransportMapping;
	stAdditionalDataIn: ST_InputTransportAdditionalData;
	// Outputs
	stStatus		: ST_OutputTransportStatus;
	stMappingOut	: ST_OutputTransportMapping;
	stAdditionaldataOut: ST_OutputTransportAdditionalData;	
END_VAR
VAR
	sNameSpaceUri			: STRING := 'urn:BeckhoffAutomation:Ua:PLC1';
	sObjectIDentifier		: STRING := 'MAIN.fbMMServer';
	sTrackServerSymbol		: STRING;
// FB's for method calls
	bCallMethod		: BOOL;
	(* Server connect *)
	fbConnectMethod			: UA_Connect;
	stConnectInfoMethod		: ST_UASessionConnectInfo;
	nConnectHdlMethod		: DWORD;
	(* Server disconnect *)
	fbDisconnectMethod	 	: UA_Disconnect;
	(* Namespace *)
	fbGetNamespaceMethod	: UA_GetNamespaceIndex;
	nNameSpaceIndexMethod	: UINT;
	(* Get/Release Method handle *)
	fbGetHandleMethod		: UA_MethodGetHandle;
	fbReleaseHandleMethod	: UA_MethodReleaseHandle;
	nHandleMethod			: DWORD;
	stObjectNodeID			: ST_UANodeID;
	stMethodNodeID			: ST_UANodeID;
	sMethodIdentifier		: STRING := '';
	(* Method call *)
	fbCallMethod			: UA_MethodCall;
	(* Declarations for state machine for method calling (OPC-UA to TrackServer) *)
	eStateMethod			: E_TrackClientState;
	eLastErrorMethodID		: E_OPC_UA_Errors;
	(* Method call data *)
	(* Input variables *)
	nNoOfInputArgs			: BYTE;
	aInputArgInfo			: ARRAY[1..10] OF ST_UAMethodArgInfo;	// change according to input parameters
	aInputData				: ARRAY[1..500] OF BYTE;				// Data area for input arguments data	
	(* Output variables *)
	nNoOfOutputArgs			: BYTE;
	aOutputArgInfo			: ARRAY[1..10] OF ST_UAMethodArgInfo; // change according to input parameters

// Method specific data structs
	stAddStationSingleData	: ST_AddStationSingleData;
	stAddStationDoubleData	: ST_AddStationDoubleData;
	stRemoveStationData		: ST_RemoveStationData;
	stEnableStationData		: ST_EnableStationData;
	stAdjustBufferPosData	: ST_AdjustBufferPosData;
	
	stGetCellIndexData		: ST_GetCellIndexData;

	stAddPathData			: ST_AddPathData;
	stRemovePathData		: ST_RemovePathData;
	stStartPathData			: ST_StartPathData;
	stResetPathData			: ST_ResetPathData;
	stSuspendPathData		: ST_SuspendPathData;
	stResumePathData		: ST_ResumePathData;

	stAddTrafficLightData	: ST_AddTrafficLightData;
	stRemoveTrafficLightData: ST_RemoveTrafficLightData;
	stTrafficLightColorData	: ST_TrafficLightColorData;
	stSetTrafficLightColorData: ST_SetTrafficLightColorData;
	
	stMoveToStationInData	: ST_MoveToStationInData;
	stMoveToStationOutData	: ST_MoveToStationOutData;
	stMoveToPositionData	: ST_MoveToPositionData;
	stMoveToBufferData		: ST_MoveToBufferData;
	stMoveToDecisionPointData: ST_MoveToDecisionPointData;
	stMoveToScannerData		: ST_MoveToScannerData;
	stMoveVehicleStatusData	: ST_MoveVehicleStatusData;
	
//	stUpdateVehicleDataData	: ST_UpdateVehicleDataData;
	stUpdateVehicleReservationDataData : ST_UpdateVehicleReservationDataData;
	stUpdateVehicleMappingDataData : ST_UpdateVehicleMappingDataData;
	stUpdateVehicleReworkDataData : ST_UpdateVehicleReworkDataData;
	stUpdateVehicleMontageData : ST_UpdateVehicleMontageData;
	stUpdateStationBufferData: ST_UpdateStationBufferData;
	stUpdateVehicleOwnerData: ST_UpdateVehicleOwnerData;
	stAddReservationData	: ST_AddReservationData;
	stRemoveReservationData	: ST_RemoveReservationData;

	stAddPathSegmentData : ST_AddPathSegmentData;
	stRemovePathSegmentData : ST_RemovePathSegmentData;
	stGetPathSegmentVehicleCountData: ST_GetPathSegmentVehicleCountData;

(* FB's for node reading *)
	(* Server connect *)
	fbConnectNodes			: UA_Connect;
	stConnectInfoNodes		: ST_UASessionConnectInfo;
	nConnectHandleNodes		: DWORD;
	(* Server disconnect *)
	fbDisconnectNodes	 	: UA_Disconnect;
	(* Namespace *)
	fbGetNamespaceNodes		: UA_GetNamespaceIndex;
	nNameSpaceIndexNodes	: UINT;
	(* Get/Release node handles *)
	fbGetHandleNodes		: UA_NodeGetHandleList;
	fbReleaseHandleNodes	: UA_NodeReleaseHandleList;
	anHandleNodes			: ARRAY [1..nMaxNodeIDsInList] OF DWORD;		// Handles to all the remote nodes
	(* Read nodes data *)
	fbReadNodes				: UA_ReadList;
	nNoOfNodes				: UINT;
	aNodeIDs				: ARRAY [1..nMaxNodeIDsInList] OF ST_UANodeID;	// Node ID's ((infor for remote variable to read)
	astNodeAddInfo			: ARRAY [1..nMaxNodeIDsInList] OF ST_UANodeAdditionalInfo;
	acbDatas				: ARRAY [1..nMaxNodeIDsInList] OF UDINT;
	cbDataTotal				: UDINT;
	eReadType				: E_OPC_NodeType;
	iReadIndex				: UINT;
	pReadNodeData			: PVOID;
	bReadDecPointVehicle	: BOOL := TRUE;	// Force reading of the vehicle at decision point before other vehicles
	bReadDecPointVehicleBusy: BOOL := FALSE;// 
	bReadDecPointCell		: BOOL;
	bReadDecPointCellDone	: BOOL;			// Used in decision point to make sure reservation data is read from cell before handling vehicle
	anExtraVehicles			: ARRAY [1..MM_MAX_NUMBER_OF_VEHICLE_ELEMENTS] OF UINT;	// Extra vehicle status data that should be read from track server
	anVehiclesToRead		: ARRAY [1..MM_MAX_NUMBER_OF_VEHICLE_ELEMENTS] OF UINT;	// Vehicles that should be read with triggered/evet-driven reading
	tonSkipPathRead			: TON;			// Skip path reading from Track Server if paths are initialized (State = Starting in M_StateMachine)
	(* Declarations for state machine for reading nodes *)
	eStateNode				: E_TrackClientState;
	tonReadInterval			: TON;
	tonErrorReset			: TON;
	rReadInterval			: REAL := 0.1;	// [S] OPC UA data polling interval
	rErrorResetDelay		: REAL := 10;	// [S] Error automatic reset time/delay
	iReadTimeMS				: UINT;
	iLastReadTimeMS			: UINT;
	(* For reading status values form Track Server *)
	abControlledPaths		: ARRAY [1..MM_MAX_NUMBER_OF_PATH_ELEMENTS] OF BOOL;		(* Paths to control from this Track Client *)
	// Index for this cell on the track server Cell status data
	iThisCellIndex			: UINT;
	iThisStationIndex		: array [1..5] of UINT;
	iStatIndex				: UINT;
// Work-Around - ADS read of status values (NOTE: Requires a route to Track Server PLC!!)
	fbReadADS				: FB_ADS_Comm;

// Status from Track Server	
	aReadVehicleData		: ARRAY [1..MM_MAX_NUMBER_OF_VEHICLE_ELEMENTS] OF ST_ReadVehicleData;
	aReadPathData			: ARRAY [1..MM_MAX_NUMBER_OF_PATH_ELEMENTS] OF ST_ReadPathData;
	aReadStationData		: ARRAY [1..MM_MAX_NUMBER_OF_STATION_ELEMENTS] OF ST_ReadStationData;
	aReadCellData			: ST_ReadCellData;
// For comparing vehicle changes
	aOldVehicleData			: ARRAY [1..MM_MAX_NUMBER_OF_VEHICLE_ELEMENTS] OF ST_StatusVehicle;
	aOldVehicleTargetReachedCnt	: ARRAY [1..MM_MAX_NUMBER_OF_VEHICLE_ELEMENTS] OF UINT;
	iOldVehicleCount		: UINT;

	// State machine
	eTrackState				: E_TrackState;
	iStationID				: UINT;
	iVehicleIndex			: UINT;
	iPathID					: UINT;
	iPathIndex				: UINT;
	bPathsOperational		: BOOL;
	bPathsSuspended			: BOOL;
	bPathsResumed			: BOOL;
	bPathsReset				: BOOL;
	tonResetTime			: TON;
	bStationData1Done		: BOOL;
	bStationData2Done		: BOOL;
	
	// Decision Point
	nDecisionPointVehicleNo	: UINT;

	// Exit point
	stExitPointSeg1LocBegin	: ST_MMLocation;	// Starting point for segment 1
	stExitPointSeg1LocEnd	: ST_MMLocation;	// Starting point for segment 1
	stExitPointSeg2LocBegin	: ST_MMLocation;	// Starting point for segment 2
	stExitPointSeg2LocEnd	: ST_MMLocation;	// Starting point for segment 2
	
	// Status generation
	iVehicle				: UINT;
	iStation				: UINT;	
	bForceVehicleUpdateOPC	: BOOL;
	
	// Command Data
	eCommandDataState		: E_CommandDataState;
	iCommandDataVehicleID	: UINT;

	// Mapping data
	eMappingDataState		: E_MappingDataState;
	iMappingDataVehicleID	: UINT;

	// Rework data
	eReworkDataState		: E_ReworkDataState;
	iReworkDataStation		: UINT;
	iReworkDataStationNo	: UINT;
	iReworkDataVehicleID	: UINT;
	sReworkDataCarrierID	: STRING(30);
	bReworkValue			: BOOL;
	
	(* Misc *)
	nOffset					: UDINT;
	bInitDone				: BOOL;
	iMethodResult			: INT;
	fbGetTime				: NT_GetTime;
//	iNodeReadErrs: UINT;
//	iNodeReads: UINT;

	// Constants
	MIN_TRACK_DIST			: REAL := 0.25;	// [m] Minimum track distance 
	
END_VAR
VAR PERSISTENT
	{attribute 'OPC.UA.DA':='1'}
	{attribute 'OPC.UA.DA.Access' := '3'}
	{attribute 'OPC.UA.DA.Description' := 'URL for OPC-UA connection to Track Server'}
	{attribute 'OPC.UA.DA.DisplayName' := 'URL for OPC-UA connection to Track Server'}
	sTrackServerUrl			: STRING := 'opc.tcp://10.38.190.130:4840';		// OPC UA address for the track server PLC
	{attribute 'OPC.UA.DA':='0'}
	sCellID					: STRING(30):= 'Cxx';							// Cell identifier
	aStations				: ARRAY [1..5] OF ST_MMStation;					// Stations
	aStationPreBufAdj		: ARRAY [1..5] OF REAL;							// Adjustment of pre-buffer positions
	aStationPostBufAdj		: ARRAY [1..5] OF REAL;							// Adjustment of post-buffer positions
	stTrafficLightLocation	: ST_MMLocation;								// Traffic light location (outlet from cell)
	stTrafficLight2Location	: ST_MMLocation;								// Traffic light location (outlet from cell)
	eCellType				: E_CellType;									// Type of station
	{attribute 'OPC.UA.DA':='1'}
	{attribute 'OPC.UA.DA.Access' := '3'}
	{attribute 'OPC.UA.DA.Description' := 'AMS NetID for ADS connection to Track Server'}
	{attribute 'OPC.UA.DA.DisplayName' := 'AMS NetID for ADS connection to Track Server'}
	sTrackServerNetID		: STRING := '10.38.190.130.1.1';				// AMS NetID of the Track Server PLC
	{attribute 'OPC.UA.DA':='0'}
	nTrackServerPortNo		: UINT := 851;									// Port number of the Track Server PLC runtime (851 = Runtime 1)
	aPaths					: ARRAY[1..MM_MAX_NUMBER_OF_PATH_ELEMENTS] OF UINT;	// Paths controlled by this cell
	{attribute 'OPC.UA.DA':='1'}
	{attribute 'OPC.UA.DA.Access' := '3'}
	{attribute 'OPC.UA.DA.Description' := 'ID of the next station on the track (where to send vehicles after DP/operation'}
	{attribute 'OPC.UA.DA.DisplayName' := 'ID of the next station on the track (where to send vehicles after DP/operation'}
	sNextStationOnTrack		: STRING(30);									// Station ID for the next station on the track
END_VAR

// Init data
M_Init();

// Handle Command Data
M_CommandData();

// Handle Mapping Data
M_MappingData();

// Handle rework data
M_ReworkData();

// State machine for method calls
M_StateMachineMethod();

// State machine for node data read
//M_StateMachineNode();
M_StateMachineNode_ADS();

// Track init state machine
M_StateMachine();

// Run worker FB's
M_Run();

// Status values
M_UpdateStatus();

// Error Warning
M_ErrorWarning();

METHOD PROTECTED M_CallAddPath : INT
VAR_INPUT
	nPathNo			: UINT;
END_VAR
IF (stAddPathData.iStatus = 2) OR (stAddPathData.iStatus = 3) THEN
	stAddPathData.iStatus := 0;
END_IF

IF (bConnectedMethod AND NOT bBusyMethod) THEN
	IF (stAddPathData.iStatus = 0) THEN
	(* Setup method calling parameters *)
		(* Method identifier *)
		sObjectIDentifier := stAddPathData.sObjectID;
		sMethodIdentifier := stAddPathData.sMethodID;
	
		(* Method Inputs *)
		stAddPathData.stInput.sCellID := sCellID;
		stAddPathData.stInput.iPath := nPathNo;
		stAddPathData.stInput.bPresent := TRUE;
		(* Fill input data area with method arguments *)
		MEMSET(ADR(aInputData), 0 ,SIZEOF(aInputData));
		nOffset := 0;
		nOffset := nOffset + MEMCPY(ADR(aInputData)+nOffset, ADR(stAddPathData.stInput), MIN(SIZEOF(stAddPathData.stInput), (SIZEOF(aInputData)-nOffset)) );
		(* Number of input arguments *)
		nNoOfInputArgs := stAddPathData.iNoOfInputArgs;
		(* Set up input argument information *)
		MEMSET(ADR(aInputArgInfo), 0, SIZEOF(aInputArgInfo));
		aInputArgInfo[1].DataType := eUAType_String;
		aInputArgInfo[1].ValueRank := -1;	// -1: Scalar 
		aInputArgInfo[1].nLenData := SIZEOF(stAddPathData.stInput.sCellID);
		aInputArgInfo[2].DataType := eUAType_UInt16;
		aInputArgInfo[2].ValueRank := -1;	// -1: Scalar 
		aInputArgInfo[2].nLenData := SIZEOF(stAddPathData.stInput.iPath);
		aInputArgInfo[3].DataType := eUAType_Boolean;
		aInputArgInfo[3].ValueRank := -1;	// -1: Scalar 
		aInputArgInfo[3].nLenData := SIZEOF(stAddPathData.stInput.bPresent);
		
		(* Method outputs *)
		(* Clear output data area *)
		(* Number of output arguments *)
		nNoOfOutputArgs := stAddPathData.iNoOfOutputArgs;
		(* Set up output argument information *)
		MEMSET(ADR(aOutputArgInfo), 0, SIZEOF(aOutputArgInfo));
		aOutputArgInfo[1].DataType := eUAType_Uint16;
		aOutputArgInfo[1].ValueRank := -1;
		aOutputArgInfo[1].nLenData := SIZEOF(stAddPathData.stOutput.eStatus);
		aOutputArgInfo[2].DataType := eUAType_String;
		aOutputArgInfo[2].ValueRank := -1;
		aOutputArgInfo[2].nLenData := SIZEOF(stAddPathData.stOutput.sMessage);
		(* Set up output  *)
		MEMSET(ADR(stAddPathData.stOutput), 0, SIZEOF(stAddPathData.stOutput));
		stAddPathData.stOutput.nNumberOfOutputArguments := nNoOfOutputArgs;
		stAddPathData.stOutput.stOutputArgInfo[1] := aOutputArgInfo[1];
		stAddPathData.stOutput.stOutputArgInfo[2] := aOutputArgInfo[2];
	
		(* Execute FB *)
		fbCallMethod.nNumberOfInputArguments := nNoOfInputArgs;
		fbCallMethod.pInputArgInfo := ADR(aInputArgInfo);
		fbCallMethod.cbInputArgInfo := (SIZEOF(aInputArgInfo[1])*nNoOfInputArgs);
		fbCallMethod.pInputArgData := ADR(aInputData);
		fbCallMethod.cbInputArgData := nOffset;
		fbCallMethod.nNumberOfOutputArguments := nNoOfOutputArgs; 
		fbCallMethod.pOutputArgInfo := ADR(aOutputArgInfo); 
		fbCallMethod.cbOutputArgInfo := (SIZEOF(aOutputArgInfo[1]) * nNoOfOutputArgs); 
		fbCallMethod.pOutputArgInfoAndData := ADR(stAddPathData.stOutput);
		fbCallMethod.cbOutputArgInfoAndData := SIZEOF(stAddPathData.stOutput);
		
		stAddPathData.iStatus := 1;
		bCallMethod := TRUE;
		
	ELSIF (stAddPathData.iStatus = 1) THEN
		// Method call Completed...
		IF (eStateMethod = E_TrackClientState.Connected) THEN
			// Method call OK
			IF (stAddPathData.stOutput.eStatus = E_MMServerStatus.eMMServerStatus_Success) THEN
				// Method returned OK
				stAddPathData.iStatus := 2;
			ELSE
				// Method returned with error
				stAddPathData.iStatus := 3;
				stAddPathData.stOutput.sMessage;
			END_IF
		ELSIF (eStateMethod = E_TrackClientState.Error) THEN
			// Method call failed
			stAddPathData.iStatus := 3;
		END_IF
		
	END_IF
END_IF

M_CallAddPath := stAddPathData.iStatus;
END_METHOD

METHOD PROTECTED M_CallAddPathSegment : INT
VAR_INPUT
	iSegmentNo		: UINT;
	nPathNo			: UINT;
	rBeginPosition	: REAL;
	rEndPosition	: REAL;
END_VAR
IF (stAddPathSegmentData.iStatus = 2) OR (stAddPathSegmentData.iStatus = 3) THEN
	stAddPathSegmentData.iStatus := 0;
END_IF

IF (bConnectedMethod AND NOT bBusyMethod) THEN
	IF (stAddPathSegmentData.iStatus = 0) THEN
	(* Setup method calling parameters *)
		(* Method identifier *)
		sObjectIDentifier := stAddPathSegmentData.sObjectID;
		sMethodIdentifier := stAddPathSegmentData.sMethodID;
	
		(* Method Inputs *)
		stAddPathSegmentData.stInput.sCellID := sCellID;
		stAddPathSegmentData.stInput.sSegmentID := CONCAT(sCellID, '_PS');
		stAddPathSegmentData.stInput.sSegmentID := CONCAT(stAddPathSegmentData.stInput.sSegmentID, UINT_TO_STRING(iSegmentNo));			
		stAddPathSegmentData.stInput.iPath := nPathNo;
		stAddPathSegmentData.stInput.rBeginPosition := rBeginPosition;
		stAddPathSegmentData.stInput.rEndPosition := rEndPosition;
		(* Fill input data area with method arguments *)
		MEMSET(ADR(aInputData), 0 ,SIZEOF(aInputData));
		nOffset := 0;
		nOffset := nOffset + MEMCPY(ADR(aInputData)+nOffset, ADR(stAddPathSegmentData.stInput), MIN(SIZEOF(stAddPathSegmentData.stInput), (SIZEOF(aInputData)-nOffset)) );
		(* Number of input arguments *)
		nNoOfInputArgs := stAddPathSegmentData.iNoOfInputArgs;
		(* Set up input argument information *)
		MEMSET(ADR(aInputArgInfo), 0, SIZEOF(aInputArgInfo));
		aInputArgInfo[1].DataType := eUAType_String;
		aInputArgInfo[1].ValueRank := -1;	// -1: Scalar 
		aInputArgInfo[1].nLenData := SIZEOF(stAddPathSegmentData.stInput.sCellID);
		aInputArgInfo[2].DataType := eUAType_String;
		aInputArgInfo[2].ValueRank := -1;	// -1: Scalar 
		aInputArgInfo[2].nLenData := SIZEOF(stAddPathSegmentData.stInput.sSegmentID);
		aInputArgInfo[3].DataType := eUAType_UInt16;
		aInputArgInfo[3].ValueRank := -1;	// -1: Scalar 
		aInputArgInfo[3].nLenData := SIZEOF(stAddPathSegmentData.stInput.iPath);
		aInputArgInfo[4].DataType := eUAType_Float;
		aInputArgInfo[4].ValueRank := -1;	// -1: Scalar 
		aInputArgInfo[4].nLenData := SIZEOF(stAddPathSegmentData.stInput.rBeginPosition);
		aInputArgInfo[5].DataType := eUAType_Float;
		aInputArgInfo[5].ValueRank := -1;	// -1: Scalar 
		aInputArgInfo[5].nLenData := SIZEOF(stAddPathSegmentData.stInput.rEndPosition);
		
		(* Method outputs *)
		(* Clear output data area *)
		(* Number of output arguments *)
		nNoOfOutputArgs := stAddPathSegmentData.iNoOfOutputArgs;
		(* Set up output argument information *)
		MEMSET(ADR(aOutputArgInfo), 0, SIZEOF(aOutputArgInfo));
		aOutputArgInfo[1].DataType := eUAType_Uint16;
		aOutputArgInfo[1].ValueRank := -1;
		aOutputArgInfo[1].nLenData := SIZEOF(stAddPathSegmentData.stOutput.eStatus);
		aOutputArgInfo[2].DataType := eUAType_String;
		aOutputArgInfo[2].ValueRank := -1;
		aOutputArgInfo[2].nLenData := SIZEOF(stAddPathSegmentData.stOutput.sMessage);
		(* Set up output  *)
		MEMSET(ADR(stAddPathSegmentData.stOutput), 0, SIZEOF(stAddPathSegmentData.stOutput));
		stAddPathSegmentData.stOutput.nNumberOfOutputArguments := nNoOfOutputArgs;
		stAddPathSegmentData.stOutput.stOutputArgInfo[1] := aOutputArgInfo[1];
		stAddPathSegmentData.stOutput.stOutputArgInfo[2] := aOutputArgInfo[2];
	
		(* Execute FB *)
		fbCallMethod.nNumberOfInputArguments := nNoOfInputArgs;
		fbCallMethod.pInputArgInfo := ADR(aInputArgInfo);
		fbCallMethod.cbInputArgInfo := (SIZEOF(aInputArgInfo[1])*nNoOfInputArgs);
		fbCallMethod.pInputArgData := ADR(aInputData);
		fbCallMethod.cbInputArgData := nOffset;
		fbCallMethod.nNumberOfOutputArguments := nNoOfOutputArgs; 
		fbCallMethod.pOutputArgInfo := ADR(aOutputArgInfo); 
		fbCallMethod.cbOutputArgInfo := (SIZEOF(aOutputArgInfo[1]) * nNoOfOutputArgs); 
		fbCallMethod.pOutputArgInfoAndData := ADR(stAddPathSegmentData.stOutput);
		fbCallMethod.cbOutputArgInfoAndData := SIZEOF(stAddPathSegmentData.stOutput);
		
		stAddPathSegmentData.iStatus := 1;
		bCallMethod := TRUE;
		
	ELSIF (stAddPathSegmentData.iStatus = 1) THEN
		// Method call Completed...
		IF (eStateMethod = E_TrackClientState.Connected) THEN
			// Method call OK
			IF (stAddPathSegmentData.stOutput.eStatus = E_MMServerStatus.eMMServerStatus_Success) THEN
				// Method returned OK
				stAddPathSegmentData.iStatus := 2;
			ELSE
				// Method returned with error
				stAddPathSegmentData.iStatus := 3;
				stAddPathSegmentData.stOutput.sMessage;
			END_IF
		ELSIF (eStateMethod = E_TrackClientState.Error) THEN
			// Method call failed
			stAddPathSegmentData.iStatus := 3;
		END_IF
		
	END_IF
END_IF

M_CallAddPathSegment := stAddPathSegmentData.iStatus;
END_METHOD

METHOD PROTECTED M_CallAddReservation : INT
VAR_INPUT
	sStationID					: STRING(30);												(* The identifier for the station. *)
	sCarrierID					: STRING(30);												(* The ID of the carrier *)
	nTicket						: UINT;														(*  *)
	nTicketSize					: UINT;														(*  *)
	nPriority					: UINT;														(*  *)
END_VAR
VAR
	i					: UINT;	
END_VAR
IF (stAddReservationData.iStatus = 2) OR (stAddReservationData.iStatus = 3) THEN
	stAddReservationData.iStatus := 0;
END_IF

IF (bConnectedMethod AND NOT bBusyMethod) THEN
	IF (stAddReservationData.iStatus = 0) THEN
	(* Setup method calling parameters *)
		(* Method identifier *)
		sObjectIDentifier := stAddReservationData.sObjectID;
		sMethodIdentifier := stAddReservationData.sMethodID;
	
		(* Method Inputs *)
		stAddReservationData.stInput.sStationID := sStationID;
		stAddReservationData.stInput.sCarrierID := sCarrierID;
		stAddReservationData.stInput.nTicket := nTicket;
		stAddReservationData.stInput.nTicketSize := nTicketSize;
		stAddReservationData.stInput.nPriority := nPriority;
		(* Fill input data area with method arguments *)
		MEMSET(ADR(aInputData), 0 ,SIZEOF(aInputData));
		nOffset := 0;
		nOffset := nOffset + MEMCPY(ADR(aInputData)+nOffset, ADR(stAddReservationData.stInput),	MIN(SIZEOF(stAddReservationData.stInput), (SIZEOF(aInputData)-nOffset)) );
		(* Number of input arguments *)
		nNoOfInputArgs := stAddReservationData.iNoOfInputArgs;
		(* Set up input argument information *)
		MEMSET(ADR(aInputArgInfo), 0, SIZEOF(aInputArgInfo));
		aInputArgInfo[1].DataType := eUAType_String;
		aInputArgInfo[1].ValueRank := -1;	// -1: Scalar 
		aInputArgInfo[1].nLenData := SIZEOF(stAddReservationData.stInput.sStationID);
		aInputArgInfo[2].DataType := eUAType_String;
		aInputArgInfo[2].ValueRank := -1;	// -1: Scalar 
		aInputArgInfo[2].nLenData := SIZEOF(stAddReservationData.stInput.sCarrierID);
		aInputArgInfo[3].DataType := eUAType_UInt16;
		aInputArgInfo[3].ValueRank := -1;	// -1: Scalar 
		aInputArgInfo[3].nLenData := SIZEOF(stAddReservationData.stInput.nTicket);
		aInputArgInfo[4].DataType := eUAType_UInt16;
		aInputArgInfo[4].ValueRank := -1;	// -1: Scalar 
		aInputArgInfo[4].nLenData := SIZEOF(stAddReservationData.stInput.nTicketSize);
		aInputArgInfo[5].DataType := eUAType_UInt16;
		aInputArgInfo[5].ValueRank := -1;	// -1: Scalar 
		aInputArgInfo[5].nLenData := SIZEOF(stAddReservationData.stInput.nPriority);
		
		(* Method outputs *)
		(* Clear output data area *)
		(* Number of output arguments *)
		nNoOfOutputArgs := stAddReservationData.iNoOfOutputArgs;
		(* Set up output argument information *)
		MEMSET(ADR(aOutputArgInfo), 0, SIZEOF(aOutputArgInfo));
		aOutputArgInfo[1].DataType := eUAType_Uint16;
		aOutputArgInfo[1].ValueRank := -1;
		aOutputArgInfo[1].nLenData := SIZEOF(stAddReservationData.stOutput.eStatus);
		aOutputArgInfo[2].DataType := eUAType_String;
		aOutputArgInfo[2].ValueRank := -1;
		aOutputArgInfo[2].nLenData := SIZEOF(stAddReservationData.stOutput.sMessage);
		(* Set up output  *)
		MEMSET(ADR(stAddReservationData.stOutput), 0, SIZEOF(stAddReservationData.stOutput));
		stAddReservationData.stOutput.nNumberOfOutputArguments := nNoOfOutputArgs;
		stAddReservationData.stOutput.stOutputArgInfo[1] := aOutputArgInfo[1];
		stAddReservationData.stOutput.stOutputArgInfo[2] := aOutputArgInfo[2];
	
		(* Execute FB *)
		fbCallMethod.nNumberOfInputArguments := nNoOfInputArgs;
		fbCallMethod.pInputArgInfo := ADR(aInputArgInfo);
		fbCallMethod.cbInputArgInfo := (SIZEOF(aInputArgInfo[1])*nNoOfInputArgs);
		fbCallMethod.pInputArgData := ADR(aInputData);
		fbCallMethod.cbInputArgData := nOffset;
		fbCallMethod.nNumberOfOutputArguments := nNoOfOutputArgs; 
		fbCallMethod.pOutputArgInfo := ADR(aOutputArgInfo); 
		fbCallMethod.cbOutputArgInfo := (SIZEOF(aOutputArgInfo[1]) * nNoOfOutputArgs); 
		fbCallMethod.pOutputArgInfoAndData := ADR(stAddReservationData.stOutput);
		fbCallMethod.cbOutputArgInfoAndData := SIZEOF(stAddReservationData.stOutput);
		
		stAddReservationData.iStatus := 1;
		bCallMethod := TRUE;
		
	ELSIF (stAddReservationData.iStatus = 1) THEN
		// Method call Completed...
		IF (eStateMethod = E_TrackClientState.Connected) THEN
			// Method call OK
			IF (stAddReservationData.stOutput.eStatus = E_MMServerStatus.eMMServerStatus_Success) THEN
				// Method returned OK
				stAddReservationData.iStatus := 2;
			ELSE
				// Method returned with error
				stAddReservationData.iStatus := 3;
				stAddReservationData.stOutput.sMessage;
			END_IF
		ELSIF (eStateMethod = E_TrackClientState.Error) THEN
			// Method call failed
			stAddReservationData.iStatus := 3;
		END_IF
		
	END_IF
END_IF

M_CallAddReservation := stAddReservationData.iStatus;
END_METHOD

METHOD PROTECTED M_CallAddStationDouble : INT
VAR_INPUT
	nStationNo			: UINT(1..5);
END_VAR
VAR
	i					: UINT;	
END_VAR
IF (stAddStationDoubleData.iStatus = 2) OR (stAddStationDoubleData.iStatus = 3) THEN
	stAddStationDoubleData.iStatus := 0;
END_IF

IF (bConnectedMethod AND NOT bBusyMethod) THEN
	IF (stAddStationDoubleData.iStatus = 0) THEN
	(* Setup method calling parameters *)
		(* Method identifier *)
		sObjectIDentifier := stAddStationDoubleData.sObjectID;
		sMethodIdentifier := stAddStationDoubleData.sMethodID;
	
		(* Method Inputs *)
		stAddStationDoubleData.stInput.sCellID := sCellID;
		stAddStationDoubleData.stInput.sID := aStations[nStationNo].sStationID;
		stAddStationDoubleData.stInput.iInPath := aStations[nStationNo].stStationData1.stLocation.nPathID;
		stAddStationDoubleData.stInput.rInPosition := aStations[nStationNo].stStationData1.stLocation.fPosition;
		stAddStationDoubleData.stInput.iOutPath := aStations[nStationNo].stStationData2.stLocation.nPathID;
		stAddStationDoubleData.stInput.rOutPosition := aStations[nStationNo].stStationData2.stLocation.fPosition;
		stAddStationDoubleData.stInput.iDecisionPath := aStations[nStationNo].stDecisionLocation.nPathID;
		stAddStationDoubleData.stInput.rDecisionPosition := aStations[nStationNo].stDecisionLocation.fPosition;
		stAddStationDoubleData.stInput.nPreBufferSize := 0;
		stAddStationDoubleData.stInput.nPostBufferSize := 0;
		// Calc buffer size
		FOR i := 1 TO 20 BY 1 DO
			IF (aStations[nStationNo].astPreBuffer[i].bPresent) THEN
				stAddStationDoubleData.stInput.nPreBufferSize := stAddStationDoubleData.stInput.nPreBufferSize + 1;
			END_IF
			IF (aStations[nStationNo].astPostBuffer[i].bPresent) THEN
				stAddStationDoubleData.stInput.nPostBufferSize := stAddStationDoubleData.stInput.nPostBufferSize + 1;
			END_IF
		END_FOR
		(* Fill input data area with method arguments *)
		MEMSET(ADR(aInputData), 0 ,SIZEOF(aInputData));
		nOffset := 0;
		nOffset := nOffset + MEMCPY(ADR(aInputData)+nOffset, ADR(stAddStationDoubleData.stInput),	MIN(SIZEOF(stAddStationDoubleData.stInput), (SIZEOF(aInputData)-nOffset)) );
		(* Number of input arguments *)
		nNoOfInputArgs := stAddStationDoubleData.iNoOfInputArgs;
		(* Set up input argument information *)
		MEMSET(ADR(aInputArgInfo), 0, SIZEOF(aInputArgInfo));
		aInputArgInfo[1].DataType := eUAType_String;
		aInputArgInfo[1].ValueRank := -1;	// -1: Scalar 
		aInputArgInfo[1].nLenData := SIZEOF(stAddStationDoubleData.stInput.sCellID);
		aInputArgInfo[2].DataType := eUAType_String;
		aInputArgInfo[2].ValueRank := -1;	// -1: Scalar 
		aInputArgInfo[2].nLenData := SIZEOF(stAddStationDoubleData.stInput.sID);
		aInputArgInfo[3].DataType := eUAType_UInt16;
		aInputArgInfo[3].ValueRank := -1;	// -1: Scalar 
		aInputArgInfo[3].nLenData := SIZEOF(stAddStationDoubleData.stInput.iInPath);
		aInputArgInfo[4].DataType := eUAType_Float;
		aInputArgInfo[4].ValueRank := -1;	// -1: Scalar 
		aInputArgInfo[4].nLenData := SIZEOF(stAddStationDoubleData.stInput.rInPosition);
		aInputArgInfo[5].DataType := eUAType_UInt16;
		aInputArgInfo[5].ValueRank := -1;	// -1: Scalar 
		aInputArgInfo[5].nLenData := SIZEOF(stAddStationDoubleData.stInput.iOutPath);
		aInputArgInfo[6].DataType := eUAType_Float;
		aInputArgInfo[6].ValueRank := -1;	// -1: Scalar 
		aInputArgInfo[6].nLenData := SIZEOF(stAddStationDoubleData.stInput.rOutPosition);
		aInputArgInfo[7].DataType := eUAType_UInt16;
		aInputArgInfo[7].ValueRank := -1;	// -1: Scalar 
		aInputArgInfo[7].nLenData := SIZEOF(stAddStationDoubleData.stInput.iDecisionPath);
		aInputArgInfo[8].DataType := eUAType_Float;
		aInputArgInfo[8].ValueRank := -1;	// -1: Scalar 
		aInputArgInfo[8].nLenData := SIZEOF(stAddStationDoubleData.stInput.rDecisionPosition);
		aInputArgInfo[9].DataType := eUAType_UInt16;
		aInputArgInfo[9].ValueRank := -1;	// -1: Scalar 
		aInputArgInfo[9].nLenData := SIZEOF(stAddStationDoubleData.stInput.nPreBufferSize);
		aInputArgInfo[10].DataType := eUAType_UInt16;
		aInputArgInfo[10].ValueRank := -1;	// -1: Scalar 
		aInputArgInfo[10].nLenData := SIZEOF(stAddStationDoubleData.stInput.nPostBufferSize);
		
		(* Method outputs *)
		(* Clear output data area *)
		(* Number of output arguments *)
		nNoOfOutputArgs := stAddStationDoubleData.iNoOfOutputArgs;
		(* Set up output argument information *)
		MEMSET(ADR(aOutputArgInfo), 0, SIZEOF(aOutputArgInfo));
		aOutputArgInfo[1].DataType := eUAType_Uint16;
		aOutputArgInfo[1].ValueRank := -1;
		aOutputArgInfo[1].nLenData := SIZEOF(stAddStationDoubleData.stOutput.eStatus);
		aOutputArgInfo[2].DataType := eUAType_String;
		aOutputArgInfo[2].ValueRank := -1;
		aOutputArgInfo[2].nLenData := SIZEOF(stAddStationDoubleData.stOutput.sMessage);
		(* Set up output  *)
		MEMSET(ADR(stAddStationDoubleData.stOutput), 0, SIZEOF(stAddStationDoubleData.stOutput));
		stAddStationDoubleData.stOutput.nNumberOfOutputArguments := nNoOfOutputArgs;
		stAddStationDoubleData.stOutput.stOutputArgInfo[1] := aOutputArgInfo[1];
		stAddStationDoubleData.stOutput.stOutputArgInfo[2] := aOutputArgInfo[2];
	
		(* Execute FB *)
		fbCallMethod.nNumberOfInputArguments := nNoOfInputArgs;
		fbCallMethod.pInputArgInfo := ADR(aInputArgInfo);
		fbCallMethod.cbInputArgInfo := (SIZEOF(aInputArgInfo[1])*nNoOfInputArgs);
		fbCallMethod.pInputArgData := ADR(aInputData);
		fbCallMethod.cbInputArgData := nOffset;
		fbCallMethod.nNumberOfOutputArguments := nNoOfOutputArgs; 
		fbCallMethod.pOutputArgInfo := ADR(aOutputArgInfo); 
		fbCallMethod.cbOutputArgInfo := (SIZEOF(aOutputArgInfo[1]) * nNoOfOutputArgs); 
		fbCallMethod.pOutputArgInfoAndData := ADR(stAddStationDoubleData.stOutput);
		fbCallMethod.cbOutputArgInfoAndData := SIZEOF(stAddStationDoubleData.stOutput);
		
		stAddStationDoubleData.iStatus := 1;
		bCallMethod := TRUE;
		
	ELSIF (stAddStationDoubleData.iStatus = 1) THEN
		// Method call Completed...
		IF (eStateMethod = E_TrackClientState.Connected) THEN
			// Method call OK
			IF (stAddStationDoubleData.stOutput.eStatus = E_MMServerStatus.eMMServerStatus_Success) THEN
				// Method returned OK
				stAddStationDoubleData.iStatus := 2;
			ELSIF (stAddStationDoubleData.stOutput.eStatus = E_MMServerStatus.eMMServerStatus_Rejected_ConfigurationAlreadyDefined) THEN
				// Method returned rejected... Already defined, this is OK
				stAddStationDoubleData.iStatus := 2;
			ELSE
				// Method returned with error
				stAddStationDoubleData.iStatus := 3;
				stAddStationDoubleData.stOutput.sMessage;
			END_IF
		ELSIF (eStateMethod = E_TrackClientState.Error) THEN
			// Method call failed
			stAddStationDoubleData.iStatus := 3;
		END_IF
		
	END_IF
END_IF

M_CallAddStationDouble := stAddStationDoubleData.iStatus;
END_METHOD

METHOD PROTECTED M_CallAddStationSingle : INT
VAR_INPUT
	nStationNo			: UINT(1..5);
END_VAR
VAR
	i					: UINT;	
END_VAR
IF (stAddStationSingleData.iStatus = 2) OR (stAddStationSingleData.iStatus = 3) THEN
	stAddStationSingleData.iStatus := 0;
END_IF

IF (bConnectedMethod AND NOT bBusyMethod) THEN
	IF (stAddStationSingleData.iStatus = 0) THEN
	(* Setup method calling parameters *)
		(* Method identifier *)
		sObjectIDentifier := stAddStationSingleData.sObjectID;
		sMethodIdentifier := stAddStationSingleData.sMethodID;
	
		(* Method Inputs *)
		stAddStationSingleData.stInput.sCellID := sCellID;
		stAddStationSingleData.stInput.sID := aStations[nStationNo].sStationID;
		stAddStationSingleData.stInput.iPath := aStations[nStationNo].stStationData1.stLocation.nPathID;
		stAddStationSingleData.stInput.rPosition := aStations[nStationNo].stStationData1.stLocation.fPosition;
		stAddStationSingleData.stInput.iDecisionPath := aStations[nStationNo].stDecisionLocation.nPathID;
		stAddStationSingleData.stInput.rDecisionPosition := aStations[nStationNo].stDecisionLocation.fPosition;
		stAddStationSingleData.stInput.nPreBufferSize := 0;
		stAddStationSingleData.stInput.nPostBufferSize := 0;
		// Calc buffer size
		FOR i := 1 TO 20 BY 1 DO
			IF (aStations[nStationNo].astPreBuffer[i].bPresent) THEN
				stAddStationSingleData.stInput.nPreBufferSize := stAddStationSingleData.stInput.nPreBufferSize + 1;
			END_IF
			IF (aStations[nStationNo].astPostBuffer[i].bPresent) THEN
				stAddStationSingleData.stInput.nPostBufferSize := stAddStationSingleData.stInput.nPostBufferSize + 1;
			END_IF
		END_FOR
		(* Fill input data area with method arguments *)
		MEMSET(ADR(aInputData), 0 ,SIZEOF(aInputData));
		nOffset := 0;
		nOffset := nOffset + MEMCPY(ADR(aInputData)+nOffset, ADR(stAddStationSingleData.stInput),	MIN(SIZEOF(stAddStationSingleData.stInput), (SIZEOF(aInputData)-nOffset)) );
		(* Number of input arguments *)
		nNoOfInputArgs := stAddStationSingleData.iNoOfInputArgs;
		(* Set up input argument information *)
		MEMSET(ADR(aInputArgInfo), 0, SIZEOF(aInputArgInfo));
		aInputArgInfo[1].DataType := eUAType_String;
		aInputArgInfo[1].ValueRank := -1;	// -1: Scalar 
		aInputArgInfo[1].nLenData := SIZEOF(stAddStationSingleData.stInput.sCellID);
		aInputArgInfo[2].DataType := eUAType_String;
		aInputArgInfo[2].ValueRank := -1;	// -1: Scalar 
		aInputArgInfo[2].nLenData := SIZEOF(stAddStationSingleData.stInput.sID);
		aInputArgInfo[3].DataType := eUAType_UInt16;
		aInputArgInfo[3].ValueRank := -1;	// -1: Scalar 
		aInputArgInfo[3].nLenData := SIZEOF(stAddStationSingleData.stInput.iPath);
		aInputArgInfo[4].DataType := eUAType_Float;
		aInputArgInfo[4].ValueRank := -1;	// -1: Scalar 
		aInputArgInfo[4].nLenData := SIZEOF(stAddStationSingleData.stInput.rPosition);
		aInputArgInfo[5].DataType := eUAType_UInt16;
		aInputArgInfo[5].ValueRank := -1;	// -1: Scalar 
		aInputArgInfo[5].nLenData := SIZEOF(stAddStationSingleData.stInput.iDecisionPath);
		aInputArgInfo[6].DataType := eUAType_Float;
		aInputArgInfo[6].ValueRank := -1;	// -1: Scalar 
		aInputArgInfo[6].nLenData := SIZEOF(stAddStationSingleData.stInput.rDecisionPosition);
		aInputArgInfo[7].DataType := eUAType_UInt16;
		aInputArgInfo[7].ValueRank := -1;	// -1: Scalar 
		aInputArgInfo[7].nLenData := SIZEOF(stAddStationSingleData.stInput.nPreBufferSize);
		aInputArgInfo[8].DataType := eUAType_UInt16;
		aInputArgInfo[8].ValueRank := -1;	// -1: Scalar 
		aInputArgInfo[8].nLenData := SIZEOF(stAddStationSingleData.stInput.nPostBufferSize);
		
		(* Method outputs *)
		(* Clear output data area *)
		(* Number of output arguments *)
		nNoOfOutputArgs := stAddStationSingleData.iNoOfOutputArgs;
		(* Set up output argument information *)
		MEMSET(ADR(aOutputArgInfo), 0, SIZEOF(aOutputArgInfo));
		aOutputArgInfo[1].DataType := eUAType_Uint16;
		aOutputArgInfo[1].ValueRank := -1;
		aOutputArgInfo[1].nLenData := SIZEOF(stAddStationSingleData.stOutput.eStatus);
		aOutputArgInfo[2].DataType := eUAType_String;
		aOutputArgInfo[2].ValueRank := -1;
		aOutputArgInfo[2].nLenData := SIZEOF(stAddStationSingleData.stOutput.sMessage);
		(* Set up output  *)
		MEMSET(ADR(stAddStationSingleData.stOutput), 0, SIZEOF(stAddStationSingleData.stOutput));
		stAddStationSingleData.stOutput.nNumberOfOutputArguments := nNoOfOutputArgs;
		stAddStationSingleData.stOutput.stOutputArgInfo[1] := aOutputArgInfo[1];
		stAddStationSingleData.stOutput.stOutputArgInfo[2] := aOutputArgInfo[2];
	
		(* Execute FB *)
		fbCallMethod.nNumberOfInputArguments := nNoOfInputArgs;
		fbCallMethod.pInputArgInfo := ADR(aInputArgInfo);
		fbCallMethod.cbInputArgInfo := (SIZEOF(aInputArgInfo[1])*nNoOfInputArgs);
		fbCallMethod.pInputArgData := ADR(aInputData);
		fbCallMethod.cbInputArgData := nOffset;
		fbCallMethod.nNumberOfOutputArguments := nNoOfOutputArgs; 
		fbCallMethod.pOutputArgInfo := ADR(aOutputArgInfo); 
		fbCallMethod.cbOutputArgInfo := (SIZEOF(aOutputArgInfo[1]) * nNoOfOutputArgs); 
		fbCallMethod.pOutputArgInfoAndData := ADR(stAddStationSingleData.stOutput);
		fbCallMethod.cbOutputArgInfoAndData := SIZEOF(stAddStationSingleData.stOutput);
		
		stAddStationSingleData.iStatus := 1;
		bCallMethod := TRUE;
		
	ELSIF (stAddStationSingleData.iStatus = 1) THEN
		// Method call Completed...
		IF (eStateMethod = E_TrackClientState.Connected) THEN
			// Method call OK
			IF (stAddStationSingleData.stOutput.eStatus = E_MMServerStatus.eMMServerStatus_Success) THEN
				// Method returned OK
				stAddStationSingleData.iStatus := 2;
			ELSIF (stAddStationSingleData.stOutput.eStatus = E_MMServerStatus.eMMServerStatus_Rejected_ConfigurationAlreadyDefined) THEN
				// Method returned rejected... Already defined, this is OK
				stAddStationSingleData.iStatus := 2;
			ELSE
				// Method returned with error
				stAddStationSingleData.iStatus := 3;
				stAddStationSingleData.stOutput.sMessage;
			END_IF
		ELSIF (eStateMethod = E_TrackClientState.Error) THEN
			// Method call failed
			stAddStationSingleData.iStatus := 3;
		END_IF
		
	END_IF
END_IF

M_CallAddStationSingle := stAddStationSingleData.iStatus;
END_METHOD

METHOD PROTECTED M_CallAddTrafficLight : INT
VAR_INPUT
	nTrafficLightID	: UINT;
	nPathID			: UINT;
	fPosition		: REAL;
END_VAR
IF (stAddTrafficLightData.iStatus = 2) OR (stAddTrafficLightData.iStatus = 3) THEN
	stAddTrafficLightData.iStatus := 0;
END_IF

IF (bConnectedMethod AND NOT bBusyMethod) THEN
	IF (stAddTrafficLightData.iStatus = 0) THEN
	(* Setup method calling parameters *)
		(* Method identifier *)
		sObjectIDentifier := stAddTrafficLightData.sObjectID;
		sMethodIdentifier := stAddTrafficLightData.sMethodID;
	
		(* Method Inputs *)
		stAddTrafficLightData.stInput.sCellID := sCellID;
		stAddTrafficLightData.stInput.sID := CONCAT(sCellID, '_TL');
		stAddTrafficLightData.stInput.sID := CONCAT(stAddTrafficLightData.stInput.sID, UINT_TO_STRING(nTrafficLightID));
		stAddTrafficLightData.stInput.iPath := nPathID;
		stAddTrafficLightData.stInput.rPosition := fPosition;
		(* Fill input data area with method arguments *)
		MEMSET(ADR(aInputData), 0 ,SIZEOF(aInputData));
		nOffset := 0;
		nOffset := nOffset + MEMCPY(ADR(aInputData)+nOffset, ADR(stAddTrafficLightData.stInput),	MIN(SIZEOF(stAddTrafficLightData.stInput),	(SIZEOF(aInputData)-nOffset)) );
		(* Number of input arguments *)
		nNoOfInputArgs := stAddTrafficLightData.iNoOfInputArgs;
		(* Set up input argument information *)
		MEMSET(ADR(aInputArgInfo), 0, SIZEOF(aInputArgInfo));
		aInputArgInfo[1].DataType := eUAType_String;
		aInputArgInfo[1].ValueRank := -1;	// -1: Scalar 
		aInputArgInfo[1].nLenData := SIZEOF(stAddTrafficLightData.stInput.sCellID);
		aInputArgInfo[2].DataType := eUAType_String;
		aInputArgInfo[2].ValueRank := -1;	// -1: Scalar 
		aInputArgInfo[2].nLenData := SIZEOF(stAddTrafficLightData.stInput.sID);
		aInputArgInfo[3].DataType := eUAType_UInt16;
		aInputArgInfo[3].ValueRank := -1;	// -1: Scalar 
		aInputArgInfo[3].nLenData := SIZEOF(stAddTrafficLightData.stInput.iPath);
		aInputArgInfo[4].DataType := eUAType_Float;
		aInputArgInfo[4].ValueRank := -1;	// -1: Scalar 
		aInputArgInfo[4].nLenData := SIZEOF(stAddTrafficLightData.stInput.rPosition);
		
		(* Method outputs *)
		(* Clear output data area *)
		(* Number of output arguments *)
		nNoOfOutputArgs := stAddTrafficLightData.iNoOfOutputArgs;
		(* Set up output argument information *)
		MEMSET(ADR(aOutputArgInfo), 0, SIZEOF(aOutputArgInfo));
		aOutputArgInfo[1].DataType := eUAType_Uint16;
		aOutputArgInfo[1].ValueRank := -1;
		aOutputArgInfo[1].nLenData := SIZEOF(stAddTrafficLightData.stOutput.eStatus);
		aOutputArgInfo[2].DataType := eUAType_String;
		aOutputArgInfo[2].ValueRank := -1;
		aOutputArgInfo[2].nLenData := SIZEOF(stAddTrafficLightData.stOutput.sMessage);
		(* Set up output  *)
		MEMSET(ADR(stAddTrafficLightData.stOutput), 0, SIZEOF(stAddTrafficLightData.stOutput));
		stAddTrafficLightData.stOutput.nNumberOfOutputArguments := nNoOfOutputArgs;
		stAddTrafficLightData.stOutput.stOutputArgInfo[1] := aOutputArgInfo[1];
		stAddTrafficLightData.stOutput.stOutputArgInfo[2] := aOutputArgInfo[2];
	
		(* Execute FB *)
		fbCallMethod.nNumberOfInputArguments := nNoOfInputArgs;
		fbCallMethod.pInputArgInfo := ADR(aInputArgInfo);
		fbCallMethod.cbInputArgInfo := (SIZEOF(aInputArgInfo[1])*nNoOfInputArgs);
		fbCallMethod.pInputArgData := ADR(aInputData);
		fbCallMethod.cbInputArgData := nOffset;
		fbCallMethod.nNumberOfOutputArguments := nNoOfOutputArgs; 
		fbCallMethod.pOutputArgInfo := ADR(aOutputArgInfo); 
		fbCallMethod.cbOutputArgInfo := (SIZEOF(aOutputArgInfo[1]) * nNoOfOutputArgs); 
		fbCallMethod.pOutputArgInfoAndData := ADR(stAddTrafficLightData.stOutput);
		fbCallMethod.cbOutputArgInfoAndData := SIZEOF(stAddTrafficLightData.stOutput);
		
		stAddTrafficLightData.iStatus := 1;
		bCallMethod := TRUE;
		
	ELSIF (stAddTrafficLightData.iStatus = 1) THEN
		// Method call Completed...
		IF (eStateMethod = E_TrackClientState.Connected) THEN
			// Method call OK
			IF (stAddTrafficLightData.stOutput.eStatus = E_MMServerStatus.eMMServerStatus_Success) THEN
				// Method returned OK
				stAddTrafficLightData.iStatus := 2;
			ELSE
				// Method returned with error
				stAddTrafficLightData.iStatus := 3;
				stAddTrafficLightData.stOutput.sMessage;
			END_IF
		ELSIF (eStateMethod = E_TrackClientState.Error) THEN
			// Method call failed
			stAddTrafficLightData.iStatus := 3;
		END_IF
		
	END_IF
END_IF

M_CallAddTrafficLight := stAddTrafficLightData.iStatus;
END_METHOD

METHOD PROTECTED M_CallAdjustBufferPosition : INT
VAR_INPUT
	nStationNo			: UINT(1..5);
	eBufferType			: E_MMStationBuffer;	// Pre- or Post-buffer
	rDistance			: REAL;					// [M9 Distance in metres (negative value to move backwards)
END_VAR
VAR
	i					: UINT;	
END_VAR
IF (stAdjustBufferPosData.iStatus = 2) OR (stAdjustBufferPosData.iStatus = 3) THEN
	stAdjustBufferPosData.iStatus := 0;
END_IF

IF (bConnectedMethod AND NOT bBusyMethod) THEN
	IF (stAdjustBufferPosData.iStatus = 0) THEN
	(* Setup method calling parameters *)
		(* Method identifier *)
		sObjectIDentifier := stAdjustBufferPosData.sObjectID;
		sMethodIdentifier := stAdjustBufferPosData.sMethodID;
	
		(* Method Inputs *)
		stAdjustBufferPosData.stInput.sStationID := aStations[nStationNo].sStationID;
		stAdjustBufferPosData.stInput.eBufferType := eBufferType;
		stAdjustBufferPosData.stInput.rDistance := rDistance;
		(* Fill input data area with method arguments *)
		MEMSET(ADR(aInputData), 0 ,SIZEOF(aInputData));
		nOffset := 0;
		nOffset := nOffset + MEMCPY(ADR(aInputData)+nOffset, ADR(stAdjustBufferPosData.stInput),	MIN(SIZEOF(stAdjustBufferPosData.stInput), (SIZEOF(aInputData)-nOffset)) );
		(* Number of input arguments *)
		nNoOfInputArgs := stAdjustBufferPosData.iNoOfInputArgs;
		(* Set up input argument information *)
		MEMSET(ADR(aInputArgInfo), 0, SIZEOF(aInputArgInfo));
		aInputArgInfo[1].DataType := eUAType_String;
		aInputArgInfo[1].ValueRank := -1;	// -1: Scalar 
		aInputArgInfo[1].nLenData := SIZEOF(stAdjustBufferPosData.stInput.sStationID);
		aInputArgInfo[2].DataType := eUAType_UInt16;
		aInputArgInfo[2].ValueRank := -1;	// -1: Scalar 
		aInputArgInfo[2].nLenData := SIZEOF(stAdjustBufferPosData.stInput.eBufferType);
		aInputArgInfo[3].DataType := eUAType_Float;
		aInputArgInfo[3].ValueRank := -1;	// -1: Scalar 
		aInputArgInfo[3].nLenData := SIZEOF(stAdjustBufferPosData.stInput.rDistance);
		
		(* Method outputs *)
		(* Clear output data area *)
		(* Number of output arguments *)
		nNoOfOutputArgs := stAdjustBufferPosData.iNoOfOutputArgs;
		(* Set up output argument information *)
		MEMSET(ADR(aOutputArgInfo), 0, SIZEOF(aOutputArgInfo));
		aOutputArgInfo[1].DataType := eUAType_Uint16;
		aOutputArgInfo[1].ValueRank := -1;
		aOutputArgInfo[1].nLenData := SIZEOF(stAdjustBufferPosData.stOutput.eStatus);
		aOutputArgInfo[2].DataType := eUAType_String;
		aOutputArgInfo[2].ValueRank := -1;
		aOutputArgInfo[2].nLenData := SIZEOF(stAdjustBufferPosData.stOutput.sMessage);
		(* Set up output  *)
		MEMSET(ADR(stAdjustBufferPosData.stOutput), 0, SIZEOF(stAdjustBufferPosData.stOutput));
		stAdjustBufferPosData.stOutput.nNumberOfOutputArguments := nNoOfOutputArgs;
		stAdjustBufferPosData.stOutput.stOutputArgInfo[1] := aOutputArgInfo[1];
		stAdjustBufferPosData.stOutput.stOutputArgInfo[2] := aOutputArgInfo[2];
	
		(* Execute FB *)
		fbCallMethod.nNumberOfInputArguments := nNoOfInputArgs;
		fbCallMethod.pInputArgInfo := ADR(aInputArgInfo);
		fbCallMethod.cbInputArgInfo := (SIZEOF(aInputArgInfo[1])*nNoOfInputArgs);
		fbCallMethod.pInputArgData := ADR(aInputData);
		fbCallMethod.cbInputArgData := nOffset;
		fbCallMethod.nNumberOfOutputArguments := nNoOfOutputArgs; 
		fbCallMethod.pOutputArgInfo := ADR(aOutputArgInfo); 
		fbCallMethod.cbOutputArgInfo := (SIZEOF(aOutputArgInfo[1]) * nNoOfOutputArgs); 
		fbCallMethod.pOutputArgInfoAndData := ADR(stAdjustBufferPosData.stOutput);
		fbCallMethod.cbOutputArgInfoAndData := SIZEOF(stAdjustBufferPosData.stOutput);
		
		stAdjustBufferPosData.iStatus := 1;
		bCallMethod := TRUE;
		
	ELSIF (stAdjustBufferPosData.iStatus = 1) THEN
		// Method call Completed...
		IF (eStateMethod = E_TrackClientState.Connected) THEN
			// Method call OK
			IF (stAdjustBufferPosData.stOutput.eStatus = E_MMServerStatus.eMMServerStatus_Success) THEN
				// Method returned OK
				stAdjustBufferPosData.iStatus := 2;
			ELSE
				// Method returned with error
				stAdjustBufferPosData.iStatus := 3;
				stAdjustBufferPosData.stOutput.sMessage;
			END_IF
		ELSIF (eStateMethod = E_TrackClientState.Error) THEN
			// Method call failed
			stAdjustBufferPosData.iStatus := 3;
		END_IF
		
	END_IF
END_IF

M_CallAdjustBufferPosition := stAdjustBufferPosData.iStatus;
END_METHOD

METHOD PROTECTED M_CallEnableStation : INT
VAR_INPUT
	nStationNo			: UINT(1..5);
END_VAR
VAR
	i					: UINT;	
END_VAR
IF (stEnableStationData.iStatus = 2) OR (stEnableStationData.iStatus = 3) THEN
	stEnableStationData.iStatus := 0;
END_IF

IF (bConnectedMethod AND NOT bBusyMethod) THEN
	IF (stEnableStationData.iStatus = 0) THEN
	(* Setup method calling parameters *)
		(* Method identifier *)
		sObjectIDentifier := stEnableStationData.sObjectID;
		sMethodIdentifier := stEnableStationData.sMethodID;
	
		(* Method Inputs *)
		stEnableStationData.stInput.sCellID := sCellID;
		stEnableStationData.stInput.sID := CONCAT(sCellID, CONCAT('_ST', UINT_TO_STRING(nStationNo)));
		stEnableStationData.stInput.bPresent := aStations[nStationNo].bPresent;
		(* Fill input data area with method arguments *)
		MEMSET(ADR(aInputData), 0 ,SIZEOF(aInputData));
		nOffset := 0;
		nOffset := nOffset + MEMCPY(ADR(aInputData)+nOffset, ADR(stEnableStationData.stInput),	MIN(SIZEOF(stEnableStationData.stInput), (SIZEOF(aInputData)-nOffset)) );
		(* Number of input arguments *)
		nNoOfInputArgs := stEnableStationData.iNoOfInputArgs;
		(* Set up input argument information *)
		MEMSET(ADR(aInputArgInfo), 0, SIZEOF(aInputArgInfo));
		aInputArgInfo[1].DataType := eUAType_String;
		aInputArgInfo[1].ValueRank := -1;	// -1: Scalar 
		aInputArgInfo[1].nLenData := SIZEOF(stEnableStationData.stInput.sCellID);
		aInputArgInfo[2].DataType := eUAType_String;
		aInputArgInfo[2].ValueRank := -1;	// -1: Scalar 
		aInputArgInfo[2].nLenData := SIZEOF(stEnableStationData.stInput.sID);
		aInputArgInfo[3].DataType := eUAType_Boolean;
		aInputArgInfo[3].ValueRank := -1;	// -1: Scalar 
		aInputArgInfo[3].nLenData := SIZEOF(stEnableStationData.stInput.bPresent);
		
		(* Method outputs *)
		(* Clear output data area *)
		(* Number of output arguments *)
		nNoOfOutputArgs := stEnableStationData.iNoOfOutputArgs;
		(* Set up output argument information *)
		MEMSET(ADR(aOutputArgInfo), 0, SIZEOF(aOutputArgInfo));
		aOutputArgInfo[1].DataType := eUAType_Uint16;
		aOutputArgInfo[1].ValueRank := -1;
		aOutputArgInfo[1].nLenData := SIZEOF(stEnableStationData.stOutput.eStatus);
		aOutputArgInfo[2].DataType := eUAType_String;
		aOutputArgInfo[2].ValueRank := -1;
		aOutputArgInfo[2].nLenData := SIZEOF(stEnableStationData.stOutput.sMessage);
		(* Set up output  *)
		MEMSET(ADR(stEnableStationData.stOutput), 0, SIZEOF(stEnableStationData.stOutput));
		stEnableStationData.stOutput.nNumberOfOutputArguments := nNoOfOutputArgs;
		stEnableStationData.stOutput.stOutputArgInfo[1] := aOutputArgInfo[1];
		stEnableStationData.stOutput.stOutputArgInfo[2] := aOutputArgInfo[2];
	
		(* Execute FB *)
		fbCallMethod.nNumberOfInputArguments := nNoOfInputArgs;
		fbCallMethod.pInputArgInfo := ADR(aInputArgInfo);
		fbCallMethod.cbInputArgInfo := (SIZEOF(aInputArgInfo[1])*nNoOfInputArgs);
		fbCallMethod.pInputArgData := ADR(aInputData);
		fbCallMethod.cbInputArgData := nOffset;
		fbCallMethod.nNumberOfOutputArguments := nNoOfOutputArgs; 
		fbCallMethod.pOutputArgInfo := ADR(aOutputArgInfo); 
		fbCallMethod.cbOutputArgInfo := (SIZEOF(aOutputArgInfo[1]) * nNoOfOutputArgs); 
		fbCallMethod.pOutputArgInfoAndData := ADR(stEnableStationData.stOutput);
		fbCallMethod.cbOutputArgInfoAndData := SIZEOF(stEnableStationData.stOutput);
		
		stEnableStationData.iStatus := 1;
		bCallMethod := TRUE;
		
	ELSIF (stEnableStationData.iStatus = 1) THEN
		// Method call Completed...
		IF (eStateMethod = E_TrackClientState.Connected) THEN
			// Method call OK
			IF (stEnableStationData.stOutput.eStatus = E_MMServerStatus.eMMServerStatus_Success) THEN
				// Method returned OK
				stEnableStationData.iStatus := 2;
			ELSE
				// Method returned with error
				stEnableStationData.iStatus := 3;
				stEnableStationData.stOutput.sMessage;
			END_IF
		ELSIF (eStateMethod = E_TrackClientState.Error) THEN
			// Method call failed
			stEnableStationData.iStatus := 3;
		END_IF
		
	END_IF
END_IF

M_CallEnableStation := stEnableStationData.iStatus;
END_METHOD

METHOD PROTECTED M_CallGetCellIndex : INT
VAR_INPUT
	sCellID				: STRING(30);
END_VAR
IF (stGetCellIndexData.iStatus = 2) OR (stGetCellIndexData.iStatus = 3) THEN
	stGetCellIndexData.iStatus := 0;
END_IF

IF (bConnectedMethod AND NOT bBusyMethod) THEN
	IF (stGetCellIndexData.iStatus = 0) THEN
	(* Setup method calling parameters *)
		(* Method identifier *)
		sObjectIDentifier := stGetCellIndexData.sObjectID;
		sMethodIdentifier := stGetCellIndexData.sMethodID;
	
		(* Method Inputs *)
		stGetCellIndexData.stInput.sCellID := sCellID;
		(* Fill input data area with method arguments *)
		MEMSET(ADR(aInputData), 0 ,SIZEOF(aInputData));
		nOffset := 0;
		nOffset := nOffset + MEMCPY(ADR(aInputData)+nOffset, ADR(stGetCellIndexData.stInput),	MIN(SIZEOF(stGetCellIndexData.stInput), (SIZEOF(aInputData)-nOffset)) );
		(* Number of input arguments *)
		nNoOfInputArgs := stGetCellIndexData.iNoOfInputArgs;
		(* Set up input argument information *)
		MEMSET(ADR(aInputArgInfo), 0, SIZEOF(aInputArgInfo));
		aInputArgInfo[1].DataType := eUAType_String;
		aInputArgInfo[1].ValueRank := -1;	// -1: Scalar 
		aInputArgInfo[1].nLenData := SIZEOF(stGetCellIndexData.stInput.sCellID);
		
		(* Method outputs *)
		(* Clear output data area *)
		(* Number of output arguments *)
		nNoOfOutputArgs := stGetCellIndexData.iNoOfOutputArgs;
		(* Set up output argument information *)
		MEMSET(ADR(aOutputArgInfo), 0, SIZEOF(aOutputArgInfo));
		aOutputArgInfo[1].DataType := eUAType_Uint16;
		aOutputArgInfo[1].ValueRank := -1;
		aOutputArgInfo[1].nLenData := SIZEOF(stGetCellIndexData.stOutput.nCellIndex);
		aOutputArgInfo[2].DataType := eUAType_Uint16;
		aOutputArgInfo[2].ValueRank := -1;
		aOutputArgInfo[2].nLenData := SIZEOF(stGetCellIndexData.stOutput.eStatus);
		aOutputArgInfo[3].DataType := eUAType_String;
		aOutputArgInfo[3].ValueRank := -1;
		aOutputArgInfo[3].nLenData := SIZEOF(stGetCellIndexData.stOutput.sMessage);
		(* Set up output  *)
		MEMSET(ADR(stGetCellIndexData.stOutput), 0, SIZEOF(stGetCellIndexData.stOutput));
		stGetCellIndexData.stOutput.nNumberOfOutputArguments := nNoOfOutputArgs;
		stGetCellIndexData.stOutput.stOutputArgInfo[1] := aOutputArgInfo[1];
		stGetCellIndexData.stOutput.stOutputArgInfo[2] := aOutputArgInfo[2];
		stGetCellIndexData.stOutput.stOutputArgInfo[3] := aOutputArgInfo[3];
	
		(* Execute FB *)
		fbCallMethod.nNumberOfInputArguments := nNoOfInputArgs;
		fbCallMethod.pInputArgInfo := ADR(aInputArgInfo);
		fbCallMethod.cbInputArgInfo := (SIZEOF(aInputArgInfo[1])*nNoOfInputArgs);
		fbCallMethod.pInputArgData := ADR(aInputData);
		fbCallMethod.cbInputArgData := nOffset;
		fbCallMethod.nNumberOfOutputArguments := nNoOfOutputArgs; 
		fbCallMethod.pOutputArgInfo := ADR(aOutputArgInfo); 
		fbCallMethod.cbOutputArgInfo := (SIZEOF(aOutputArgInfo[1]) * nNoOfOutputArgs); 
		fbCallMethod.pOutputArgInfoAndData := ADR(stGetCellIndexData.stOutput);
		fbCallMethod.cbOutputArgInfoAndData := SIZEOF(stGetCellIndexData.stOutput);
		
		stGetCellIndexData.iStatus := 1;
		bCallMethod := TRUE;
		
	ELSIF (stGetCellIndexData.iStatus = 1) THEN
		// Method call Completed...
		IF (eStateMethod = E_TrackClientState.Connected) THEN
			// Method call OK
			IF (stGetCellIndexData.stOutput.eStatus = E_MMServerStatus.eMMServerStatus_Success) THEN
				// Method returned OK
				stGetCellIndexData.iStatus := 2;
			ELSE
				// Method returned with error
				stGetCellIndexData.iStatus := 3;
				stGetCellIndexData.stOutput.sMessage;
			END_IF
		ELSIF (eStateMethod = E_TrackClientState.Error) THEN
			// Method call failed
			stGetCellIndexData.iStatus := 3;
		END_IF
		
	END_IF
END_IF

M_CallGetCellIndex := stGetCellIndexData.iStatus;
END_METHOD

METHOD PROTECTED M_CallGetPathSegmentVehicleCount : INT
VAR_INPUT
	iSegmentNo		: UINT;
END_VAR
IF (stGetPathSegmentVehicleCountData.iStatus = 2) OR (stGetPathSegmentVehicleCountData.iStatus = 3) THEN
	stGetPathSegmentVehicleCountData.iStatus := 0;
END_IF

IF (bConnectedMethod AND NOT bBusyMethod) THEN
	IF (stGetPathSegmentVehicleCountData.iStatus = 0) THEN
	(* Setup method calling parameters *)
		(* Method identifier *)
		sObjectIDentifier := stGetPathSegmentVehicleCountData.sObjectID;
		sMethodIdentifier := stGetPathSegmentVehicleCountData.sMethodID;
	
		(* Method Inputs *)
		stGetPathSegmentVehicleCountData.stInput.sCellID := sCellID;
		stGetPathSegmentVehicleCountData.stInput.sSegmentID := CONCAT(sCellID, '_PS');
		stGetPathSegmentVehicleCountData.stInput.sSegmentID := CONCAT(stGetPathSegmentVehicleCountData.stInput.sSegmentID, UINT_TO_STRING(iSegmentNo));			
		(* Fill input data area with method arguments *)
		MEMSET(ADR(aInputData), 0 ,SIZEOF(aInputData));
		nOffset := 0;
		nOffset := nOffset + MEMCPY(ADR(aInputData)+nOffset, ADR(stGetPathSegmentVehicleCountData.stInput),	MIN(SIZEOF(stGetPathSegmentVehicleCountData.stInput), (SIZEOF(aInputData)-nOffset)) );
		(* Number of input arguments *)
		nNoOfInputArgs := stGetPathSegmentVehicleCountData.iNoOfInputArgs;
		(* Set up input argument information *)
		MEMSET(ADR(aInputArgInfo), 0, SIZEOF(aInputArgInfo));
		aInputArgInfo[1].DataType := eUAType_String;
		aInputArgInfo[1].ValueRank := -1;	// -1: Scalar 
		aInputArgInfo[1].nLenData := SIZEOF(stGetPathSegmentVehicleCountData.stInput.sCellID);
		aInputArgInfo[2].DataType := eUAType_String;
		aInputArgInfo[2].ValueRank := -1;	// -1: Scalar 
		aInputArgInfo[2].nLenData := SIZEOF(stGetPathSegmentVehicleCountData.stInput.sSegmentID);
		
		(* Method outputs *)
		(* Clear output data area *)
		(* Number of output arguments *)
		nNoOfOutputArgs := stGetPathSegmentVehicleCountData.iNoOfOutputArgs;
		(* Set up output argument information *)
		MEMSET(ADR(aOutputArgInfo), 0, SIZEOF(aOutputArgInfo));
		aOutputArgInfo[1].DataType := eUAType_Uint16;
		aOutputArgInfo[1].ValueRank := -1;
		aOutputArgInfo[1].nLenData := SIZEOF(stGetPathSegmentVehicleCountData.stOutput.iVehicleCount);
		aOutputArgInfo[2].DataType := eUAType_Uint16;
		aOutputArgInfo[2].ValueRank := -1;
		aOutputArgInfo[2].nLenData := SIZEOF(stGetPathSegmentVehicleCountData.stOutput.eStatus);
		aOutputArgInfo[3].DataType := eUAType_String;
		aOutputArgInfo[3].ValueRank := -1;
		aOutputArgInfo[3].nLenData := SIZEOF(stGetPathSegmentVehicleCountData.stOutput.sMessage);
		(* Set up output  *)
		MEMSET(ADR(stGetPathSegmentVehicleCountData.stOutput), 0, SIZEOF(stGetPathSegmentVehicleCountData.stOutput));
		stGetPathSegmentVehicleCountData.stOutput.nNumberOfOutputArguments := nNoOfOutputArgs;
		stGetPathSegmentVehicleCountData.stOutput.stOutputArgInfo[1] := aOutputArgInfo[1];
		stGetPathSegmentVehicleCountData.stOutput.stOutputArgInfo[2] := aOutputArgInfo[2];
		stGetPathSegmentVehicleCountData.stOutput.stOutputArgInfo[3] := aOutputArgInfo[3];
	
		(* Execute FB *)
		fbCallMethod.nNumberOfInputArguments := nNoOfInputArgs;
		fbCallMethod.pInputArgInfo := ADR(aInputArgInfo);
		fbCallMethod.cbInputArgInfo := (SIZEOF(aInputArgInfo[1])*nNoOfInputArgs);
		fbCallMethod.pInputArgData := ADR(aInputData);
		fbCallMethod.cbInputArgData := nOffset;
		fbCallMethod.nNumberOfOutputArguments := nNoOfOutputArgs; 
		fbCallMethod.pOutputArgInfo := ADR(aOutputArgInfo); 
		fbCallMethod.cbOutputArgInfo := (SIZEOF(aOutputArgInfo[1]) * nNoOfOutputArgs);
		fbCallMethod.pOutputArgInfoAndData := ADR(stGetPathSegmentVehicleCountData.stOutput);
		fbCallMethod.cbOutputArgInfoAndData := SIZEOF(stGetPathSegmentVehicleCountData.stOutput);
		
		stGetPathSegmentVehicleCountData.iStatus := 1;
		bCallMethod := TRUE;
		
	ELSIF (stGetPathSegmentVehicleCountData.iStatus = 1) THEN
		// Method call Completed...
		IF (eStateMethod = E_TrackClientState.Connected) THEN
			// Method call OK
			IF (stGetPathSegmentVehicleCountData.stOutput.eStatus = E_MMServerStatus.eMMServerStatus_Success) THEN
				// Method returned OK
				stGetPathSegmentVehicleCountData.iStatus := 2;
			ELSE
				// Method returned with error
				stGetPathSegmentVehicleCountData.iStatus := 3;
				stGetPathSegmentVehicleCountData.stOutput.sMessage;
			END_IF
		ELSIF (eStateMethod = E_TrackClientState.Error) THEN
			// Method call failed
			stGetPathSegmentVehicleCountData.iStatus := 3;
		END_IF
		
	END_IF
END_IF

M_CallGetPathSegmentVehicleCount := stGetPathSegmentVehicleCountData.iStatus;
END_METHOD

METHOD PROTECTED M_CallMoveVehicleStatus : INT
VAR_INPUT
	iCommandID		: UINT;
END_VAR
VAR_OUTPUT
	eMoveStatus		: E_VehicleMoveState := E_VehicleMoveState.Unknown;
END_VAR
IF (stMoveVehicleStatusData.iStatus = 2) OR (stMoveVehicleStatusData.iStatus = 3) THEN
	stMoveVehicleStatusData.iStatus := 0;
END_IF

IF (bConnectedMethod AND NOT bBusyMethod) THEN
	IF (stMoveVehicleStatusData.iStatus = 0) THEN
	(* Setup method calling parameters *)
		(* Method identifier *)
		sObjectIDentifier := stMoveVehicleStatusData.sObjectID;
		sMethodIdentifier := stMoveVehicleStatusData.sMethodID;
	
		(* Method Inputs *)
		stMoveVehicleStatusData.stInput.iCommandID := iCommandID;
		(* Fill input data area with method arguments *)
		MEMSET(ADR(aInputData), 0 ,SIZEOF(aInputData));
		nOffset := 0;
		nOffset := nOffset + MEMCPY(ADR(aInputData)+nOffset, ADR(stMoveVehicleStatusData.stInput),	MIN(SIZEOF(stMoveVehicleStatusData.stInput), (SIZEOF(aInputData)-nOffset)) );
		(* Number of input arguments *)
		nNoOfInputArgs := stMoveVehicleStatusData.iNoOfInputArgs;
		(* Set up input argument information *)
		MEMSET(ADR(aInputArgInfo), 0, SIZEOF(aInputArgInfo));
		aInputArgInfo[1].DataType := eUAType_UInt16;
		aInputArgInfo[1].ValueRank := -1;	// -1: Scalar 
		aInputArgInfo[1].nLenData := SIZEOF(stMoveVehicleStatusData.stInput.iCommandID);
		
		(* Method outputs *)
		(* Clear output data area *)
		(* Number of output arguments *)
		nNoOfOutputArgs := stMoveVehicleStatusData.iNoOfOutputArgs;
		(* Set up output argument information *)
		MEMSET(ADR(aOutputArgInfo), 0, SIZEOF(aOutputArgInfo));
		aOutputArgInfo[1].DataType := eUAType_Uint16;
		aOutputArgInfo[1].ValueRank := -1;
		aOutputArgInfo[1].nLenData := SIZEOF(stMoveVehicleStatusData.stOutput.eStatus);
		aOutputArgInfo[2].DataType := eUAType_String;
		aOutputArgInfo[2].ValueRank := -1;
		aOutputArgInfo[2].nLenData := SIZEOF(stMoveVehicleStatusData.stOutput.sMessage);
		aOutputArgInfo[3].DataType := eUAType_UInt16;
		aOutputArgInfo[3].ValueRank := -1;
		aOutputArgInfo[3].nLenData := SIZEOF(stMoveVehicleStatusData.stOutput.eMoveStatus);
		(* Set up output  *)
		MEMSET(ADR(stMoveVehicleStatusData.stOutput), 0, SIZEOF(stMoveVehicleStatusData.stOutput));
		stMoveVehicleStatusData.stOutput.nNumberOfOutputArguments := nNoOfOutputArgs;
		stMoveVehicleStatusData.stOutput.stOutputArgInfo[1] := aOutputArgInfo[1];
		stMoveVehicleStatusData.stOutput.stOutputArgInfo[2] := aOutputArgInfo[2];
		stMoveVehicleStatusData.stOutput.stOutputArgInfo[3] := aOutputArgInfo[3];
	
		(* Execute FB *)
		fbCallMethod.nNumberOfInputArguments := nNoOfInputArgs;
		fbCallMethod.pInputArgInfo := ADR(aInputArgInfo);
		fbCallMethod.cbInputArgInfo := (SIZEOF(aInputArgInfo[1])*nNoOfInputArgs);
		fbCallMethod.pInputArgData := ADR(aInputData);
		fbCallMethod.cbInputArgData := nOffset;
		fbCallMethod.nNumberOfOutputArguments := nNoOfOutputArgs; 
		fbCallMethod.pOutputArgInfo := ADR(aOutputArgInfo); 
		fbCallMethod.cbOutputArgInfo := (SIZEOF(aOutputArgInfo[1]) * nNoOfOutputArgs); 
		fbCallMethod.pOutputArgInfoAndData := ADR(stMoveVehicleStatusData.stOutput);
		fbCallMethod.cbOutputArgInfoAndData := SIZEOF(stMoveVehicleStatusData.stOutput);
		
		stMoveVehicleStatusData.iStatus := 1;
		bCallMethod := TRUE;
		
	ELSIF (stMoveVehicleStatusData.iStatus = 1) THEN
		// Method call Completed...
		IF (iCommandID = stMoveVehicleStatusData.stInput.iCommandID) THEN
			// Correct Command ID!
			IF (eStateMethod = E_TrackClientState.Connected) THEN
				// Method call OK
				IF (stMoveVehicleStatusData.stOutput.eStatus = E_MMServerStatus.eMMServerStatus_Success) THEN
					// Method returned OK
					stMoveVehicleStatusData.iStatus := 2;
					eMoveStatus := stMoveVehicleStatusData.stOutput.eMoveStatus;
					
				ELSE
					// Method returned with error
					stMoveVehicleStatusData.iStatus := 3;
					stMoveVehicleStatusData.stOutput.sMessage;
					stMoveVehicleStatusData.stOutput.eStatus;
	
				END_IF
	
			ELSIF (eStateMethod = E_TrackClientState.Error) THEN
				// Method call failed
				stMoveVehicleStatusData.iStatus := 3;
			END_IF

		ELSE
			// Do not allow to return 2 (or 3) if the CommandID is not the same as the movment was started with!
			F_LogLine('TC_VS: Wrong Command ID (%d)', iCommandID);
			
		END_IF
		
	END_IF

END_IF

M_CallMoveVehicleStatus := stMoveVehicleStatusData.iStatus;
END_METHOD

METHOD PROTECTED M_CallMoveVehicleToBuffer : INT
VAR_INPUT
	eInputType			: E_MMVehicleInputType;
	sInput				: STRING;
	sStationID			: STRING;
	eBufferType			: E_MMStationBuffer;
	nBufferIndex		: USINT;
	eDirection			: E_MMDirection := E_MMDirection.eMMDirection_Forward;	// Default forward direction
	fVelocity			: REAL;
	fAcceleration		: REAL;
END_VAR
VAR
	i					: UINT;	
	nPostBufferSize: INT;
END_VAR
VAR_OUTPUT
	iCmdID				: UINT;
END_VAR
IF (stMoveToBufferData.iStatus = 2) OR (stMoveToBufferData.iStatus = 3) THEN
	stMoveToBufferData.iStatus := 0;
END_IF

IF (bConnectedMethod AND NOT bBusyMethod) THEN
	IF (stMoveToBufferData.iStatus = 0) THEN
	(* Setup method calling parameters *)
		(* Method identifier *)
		sObjectIDentifier := stMoveToBufferData.sObjectID;
		sMethodIdentifier := stMoveToBufferData.sMethodID;
	
		(* Method Inputs *)
		stMoveToBufferData.stInput.eInputType := eInputType;
		stMoveToBufferData.stInput.sInput := sInput;
		stMoveToBufferData.stInput.sStationID := sStationID;
		stMoveToBufferData.stInput.eStationBufferType := eBufferType;
		stMoveToBufferData.stInput.nIndex := nBufferIndex;
		stMoveToBufferData.stInput.eDirection := eDirection;
		stMoveToBufferData.stInput.nFollowID := 0;
		stMoveToBufferData.stInput.fVelocity := fVelocity;
		stMoveToBufferData.stInput.fAcceleration := fAcceleration;
		
